	            END_IF;
	            IF NOT #iqUDT_WorkstationStatus."170".PEC_EoS.PEC THEN
	                IF #sa_TrackingArray_170[#iqUDT_Configuration."170".PEC_EoS.Distance / 10 - 2] > #iqUDT_Configuration.GlobalConfig.GINRangeStart
	                    AND #sa_TrackingArray_170[#iqUDT_Configuration."170".PEC_EoS.Distance / 10 - 2] < ((#iqUDT_Configuration.GlobalConfig.GINRangeStart + #iqUDT_Configuration.GlobalConfig.GINRangeEnd) / 2) THEN
	                    IF #si_EmptyBinRequiredCounter1X0 > 0 THEN
	                        #si_EmptyBinRequiredCounter1X0 -= 1;
	                    END_IF;
	                ELSE

	                    IF #si_PartialyBinRequiredCounter1X0 > 0 THEN
	                        #si_PartialyBinRequiredCounter1X0 -= 1;
	                    ELSE
	                        IF #si_EmptyBinRequiredCounter1X0 > 0 THEN
	                            #si_EmptyBinRequiredCounter1X0 -= 1;
	                        END_IF;


	                    END_IF;

	                END_IF;


	            END_IF; *)


	        END_REGION

	    END_REGION

	    REGION Barcode handling

	        REGION 050

	            IF #iqUDT_WorkstationCommonStatus."050".Dieback
	                AND NOT #iqUDT_WorkstationStatus."050".PEC_EoS.PEC
	                AND #sa_TrackingArray_050[(#iqUDT_Configuration."050".PEC_EoS.Distance / 10) - 1] > 0
	            THEN

	                IF #iqUDT_FirstWESInterface.Field[1].WES2PLC.SetContainerID THEN

	                    "DB_GIN".GIN[#sa_TrackingArray_050[(#iqUDT_Configuration."050".PEC_EoS.Distance / 10) - 1]].General.Identification.Barcode := #iqUDT_FirstWESInterface.Field[1].WES2PLC.ContainerID;
	                    #iqUDT_FirstWESInterface.Field[1].WES2PLC.SetContainerID := 0;

	                END_IF;

	                IF #iqUDT_FirstWESInterface.Field[1].PLC2WES.ContainerID <> "DB_GIN".GIN[#sa_TrackingArray_050[(#iqUDT_Configuration."050".PEC_EoS.Distance / 10) - 1]].General.Identification.Barcode
	                THEN

	                    #iqUDT_FirstWESInterface.Field[1].PLC2WES.ContainerID := "DB_GIN".GIN[#sa_TrackingArray_050[(#iqUDT_Configuration."050".PEC_EoS.Distance / 10) - 1]].General.Identification.Barcode;
	                    #iqUDT_FirstWESInterface.Field[1].PLC2WES.SetContainerID := TRUE;
	                END_IF;
	            ELSE
	                IF #iqUDT_FirstWESInterface.Field[1].PLC2WES.ContainerID <> #cs_MissingBarcodeCode
	                THEN
	                    #iqUDT_FirstWESInterface.Field[1].PLC2WES.ContainerID := #cs_MissingBarcodeCode;
	                    #iqUDT_FirstWESInterface.Field[1].PLC2WES.SetContainerID := TRUE;
	                END_IF;

	            END_IF;

	        END_REGION

	        REGION 060

	            IF #iqUDT_WorkstationCommonStatus."060".Dieback
	                AND NOT #iqUDT_WorkstationStatus."060".PEC_EoS.PEC
	                AND #sa_TrackingArray_060[(#iqUDT_Configuration."060".PEC_EoS.Distance / 10) - 1] > 0
	            THEN

	                IF #iqUDT_FirstWESInterface.Field[2].WES2PLC.SetContainerID THEN

	                    "DB_GIN".GIN[#sa_TrackingArray_060[(#iqUDT_Configuration."060".PEC_EoS.Distance / 10) - 1]].General.Identification.Barcode := #iqUDT_FirstWESInterface.Field[2].WES2PLC.ContainerID;
	                    #iqUDT_FirstWESInterface.Field[2].WES2PLC.SetContainerID := 0;

	                END_IF;

	                IF #iqUDT_FirstWESInterface.Field[2].PLC2WES.ContainerID <> "DB_GIN".GIN[#sa_TrackingArray_060[(#iqUDT_Configuration."060".PEC_EoS.Distance / 10) - 1]].General.Identification.Barcode
	                THEN

	                    #iqUDT_FirstWESInterface.Field[2].PLC2WES.ContainerID := "DB_GIN".GIN[#sa_TrackingArray_060[(#iqUDT_Configuration."060".PEC_EoS.Distance / 10) - 1]].General.Identification.Barcode;
	                    #iqUDT_FirstWESInterface.Field[2].PLC2WES.SetContainerID := TRUE;
	                END_IF;
	            ELSE
	                IF #iqUDT_FirstWESInterface.Field[2].PLC2WES.ContainerID <> #cs_MissingBarcodeCode
	                THEN
	                    #iqUDT_FirstWESInterface.Field[2].PLC2WES.ContainerID := #cs_MissingBarcodeCode;
	                    #iqUDT_FirstWESInterface.Field[2].PLC2WES.SetContainerID := TRUE;
	                END_IF;

	            END_IF;

	        END_REGION

	        REGION 070

	            IF #iqUDT_WorkstationCommonStatus."070".Dieback
	                AND NOT #iqUDT_WorkstationStatus."070".PEC_EoS.PEC
	                AND #sa_TrackingArray_070[(#iqUDT_Configuration."070".PEC_EoS.Distance / 10) - 1] > 0
	            THEN

	                IF #iqUDT_FirstWESInterface.Field[3].WES2PLC.SetContainerID THEN

	                    "DB_GIN".GIN[#sa_TrackingArray_070[(#iqUDT_Configuration."070".PEC_EoS.Distance / 10) - 1]].General.Identification.Barcode := #iqUDT_FirstWESInterface.Field[3].WES2PLC.ContainerID;
	                    #iqUDT_FirstWESInterface.Field[3].WES2PLC.SetContainerID := 0;

	                END_IF;

	                IF #iqUDT_FirstWESInterface.Field[3].PLC2WES.ContainerID <> "DB_GIN".GIN[#sa_TrackingArray_070[(#iqUDT_Configuration."070".PEC_EoS.Distance / 10) - 1]].General.Identification.Barcode
	                THEN

	                    #iqUDT_FirstWESInterface.Field[3].PLC2WES.ContainerID := "DB_GIN".GIN[#sa_TrackingArray_070[(#iqUDT_Configuration."070".PEC_EoS.Distance / 10) - 1]].General.Identification.Barcode;
	                    #iqUDT_FirstWESInterface.Field[3].PLC2WES.SetContainerID := TRUE;
	                END_IF;
	            ELSE
	                IF #iqUDT_FirstWESInterface.Field[3].PLC2WES.ContainerID <> #cs_MissingBarcodeCode
	                THEN
	                    #iqUDT_FirstWESInterface.Field[3].PLC2WES.ContainerID := #cs_MissingBarcodeCode;
	                    #iqUDT_FirstWESInterface.Field[3].PLC2WES.SetContainerID := TRUE;
	                END_IF;

	            END_IF;

	        END_REGION


	        REGION 150

	            IF #iqUDT_WorkstationCommonStatus."150".Dieback
	                AND NOT #iqUDT_WorkstationStatus."150".PEC_EoS.PEC
	                AND #sa_TrackingArray_150[(#iqUDT_Configuration."150".PEC_EoS.Distance / 10) - 1] > 0
	            THEN

	                IF #iqUDT_SecondWESInterface.Field[1].WES2PLC.SetContainerID THEN

	                    "DB_GIN".GIN[#sa_TrackingArray_150[(#iqUDT_Configuration."150".PEC_EoS.Distance / 10) - 1]].General.Identification.Barcode := #iqUDT_SecondWESInterface.Field[1].WES2PLC.ContainerID;
	                    #iqUDT_SecondWESInterface.Field[1].WES2PLC.SetContainerID := 0;

	                END_IF;

	                IF #iqUDT_SecondWESInterface.Field[1].PLC2WES.ContainerID <> "DB_GIN".GIN[#sa_TrackingArray_150[(#iqUDT_Configuration."150".PEC_EoS.Distance / 10) - 1]].General.Identification.Barcode
	                THEN

	                    #iqUDT_SecondWESInterface.Field[1].PLC2WES.ContainerID := "DB_GIN".GIN[#sa_TrackingArray_150[(#iqUDT_Configuration."150".PEC_EoS.Distance / 10) - 1]].General.Identification.Barcode;
	                    #iqUDT_SecondWESInterface.Field[1].PLC2WES.SetContainerID := TRUE;
	                END_IF;
	            ELSE
	                IF #iqUDT_SecondWESInterface.Field[1].PLC2WES.ContainerID <> #cs_MissingBarcodeCode
	                THEN
	                    #iqUDT_SecondWESInterface.Field[1].PLC2WES.ContainerID := #cs_MissingBarcodeCode;
	                    #iqUDT_SecondWESInterface.Field[1].PLC2WES.SetContainerID := TRUE;
	                END_IF;

	            END_IF;

	        END_REGION

	        REGION 160

	            IF #iqUDT_WorkstationCommonStatus."160".Dieback
	                AND NOT #iqUDT_WorkstationStatus."160".PEC_EoS.PEC
	                AND #sa_TrackingArray_160[(#iqUDT_Configuration."160".PEC_EoS.Distance / 10) - 1] > 0
	            THEN

	                IF #iqUDT_SecondWESInterface.Field[2].WES2PLC.SetContainerID THEN

	                    "DB_GIN".GIN[#sa_TrackingArray_160[(#iqUDT_Configuration."160".PEC_EoS.Distance / 10) - 1]].General.Identification.Barcode := #iqUDT_SecondWESInterface.Field[2].WES2PLC.ContainerID;
	                    #iqUDT_SecondWESInterface.Field[2].WES2PLC.SetContainerID := 0;

	                END_IF;

	                IF #iqUDT_SecondWESInterface.Field[2].PLC2WES.ContainerID <> "DB_GIN".GIN[#sa_TrackingArray_160[(#iqUDT_Configuration."160".PEC_EoS.Distance / 10) - 1]].General.Identification.Barcode
	                THEN

	                    #iqUDT_SecondWESInterface.Field[2].PLC2WES.ContainerID := "DB_GIN".GIN[#sa_TrackingArray_160[(#iqUDT_Configuration."160".PEC_EoS.Distance / 10) - 1]].General.Identification.Barcode;
	                    #iqUDT_SecondWESInterface.Field[2].PLC2WES.SetContainerID := TRUE;
	                END_IF;
	            ELSE
	                IF #iqUDT_SecondWESInterface.Field[2].PLC2WES.ContainerID <> #cs_MissingBarcodeCode
	                THEN
	                    #iqUDT_SecondWESInterface.Field[2].PLC2WES.ContainerID := #cs_MissingBarcodeCode;
	                    #iqUDT_SecondWESInterface.Field[2].PLC2WES.SetContainerID := TRUE;
	                END_IF;

	            END_IF;

	        END_REGION

	        REGION 170

	            IF #iqUDT_WorkstationCommonStatus."170".Dieback
	                AND NOT #iqUDT_WorkstationStatus."170".PEC_EoS.PEC
	                AND #sa_TrackingArray_170[(#iqUDT_Configuration."170".PEC_EoS.Distance / 10) - 1] > 0
	            THEN

	                IF #iqUDT_SecondWESInterface.Field[3].WES2PLC.SetContainerID THEN

	                    "DB_GIN".GIN[#sa_TrackingArray_170[(#iqUDT_Configuration."170".PEC_EoS.Distance / 10) - 1]].General.Identification.Barcode := #iqUDT_SecondWESInterface.Field[3].WES2PLC.ContainerID;
	                    #iqUDT_SecondWESInterface.Field[3].WES2PLC.SetContainerID := 0;

	                END_IF;

	                IF #iqUDT_SecondWESInterface.Field[3].PLC2WES.ContainerID <> "DB_GIN".GIN[#sa_TrackingArray_170[(#iqUDT_Configuration."170".PEC_EoS.Distance / 10) - 1]].General.Identification.Barcode
	                THEN

	                    #iqUDT_SecondWESInterface.Field[3].PLC2WES.ContainerID := "DB_GIN".GIN[#sa_TrackingArray_170[(#iqUDT_Configuration."170".PEC_EoS.Distance / 10) - 1]].General.Identification.Barcode;
	                    #iqUDT_SecondWESInterface.Field[3].PLC2WES.SetContainerID := TRUE;
	                END_IF;
	            ELSE
	                IF #iqUDT_SecondWESInterface.Field[3].PLC2WES.ContainerID <> #cs_MissingBarcodeCode
	                THEN
	                    #iqUDT_SecondWESInterface.Field[3].PLC2WES.ContainerID := #cs_MissingBarcodeCode;
	                    #iqUDT_SecondWESInterface.Field[3].PLC2WES.SetContainerID := TRUE;
	                END_IF;

	            END_IF;

	        END_REGION


	    END_REGION

	    REGION Clearing tracking

	        IF (#sx_Hold050
	            AND #sa_TrackingArray_050[(#iqUDT_Configuration."050".PEC_EoS.Distance - 10) / 10] <> 0
	            AND #iqUDT_WorkstationStatus."050".PEC_EoS.PEC)

	        THEN

	            #tx_ArraySize := "FC_GetNrOfArrayEl"(#sa_TrackingArray_050);

	            FILL_BLK(IN    := 0,
	                     COUNT := INT_TO_ULINT(#tx_ArraySize),
	                     OUT   => #sa_TrackingArray_050[0]);

	        END_IF;

	        IF (#sx_Hold060
	            AND #sa_TrackingArray_060[(#iqUDT_Configuration."060".PEC_EoS.Distance - 10) / 10] <> 0
	            AND #iqUDT_WorkstationStatus."060".PEC_EoS.PEC)

	        THEN

	            #tx_ArraySize := "FC_GetNrOfArrayEl"(#sa_TrackingArray_060);

	            FILL_BLK(IN    := 0,
	                     COUNT := INT_TO_ULINT(#tx_ArraySize),
	                     OUT   => #sa_TrackingArray_060[0]);

	        END_IF;

	        IF (#sx_Hold070
	            AND #sa_TrackingArray_070[(#iqUDT_Configuration."070".PEC_EoS.Distance - 10) / 10] <> 0
	            AND #iqUDT_WorkstationStatus."070".PEC_EoS.PEC)

	        THEN

	            #tx_ArraySize := "FC_GetNrOfArrayEl"(#sa_TrackingArray_070);

	            FILL_BLK(IN    := 0,
	                     COUNT := INT_TO_ULINT(#tx_ArraySize),
	                     OUT   => #sa_TrackingArray_070[0]);

	        END_IF;


	        IF (#sx_Hold150
	            AND #sa_TrackingArray_150[(#iqUDT_Configuration."150".PEC_EoS.Distance - 10) / 10] <> 0
	            AND #iqUDT_WorkstationStatus."150".PEC_EoS.PEC)

	        THEN

	            #tx_ArraySize := "FC_GetNrOfArrayEl"(#sa_TrackingArray_150);

	            FILL_BLK(IN    := 0,
	                     COUNT := INT_TO_ULINT(#tx_ArraySize),
	                     OUT   => #sa_TrackingArray_150[0]);

	        END_IF;

	        IF (#sx_Hold160
	            AND #sa_TrackingArray_160[(#iqUDT_Configuration."160".PEC_EoS.Distance - 10) / 10] <> 0
	            AND #iqUDT_WorkstationStatus."160".PEC_EoS.PEC)

	        THEN

	            #tx_ArraySize := "FC_GetNrOfArrayEl"(#sa_TrackingArray_160);

	            FILL_BLK(IN    := 0,
	                     COUNT := INT_TO_ULINT(#tx_ArraySize),
	                     OUT   => #sa_TrackingArray_060[0]);

	        END_IF;

	        IF (#sx_Hold170
	            AND #sa_TrackingArray_170[(#iqUDT_Configuration."170".PEC_EoS.Distance - 10) / 10] <> 0
	            AND #iqUDT_WorkstationStatus."170".PEC_EoS.PEC)

	        THEN

	            #tx_ArraySize := "FC_GetNrOfArrayEl"(#sa_TrackingArray_170);

	            FILL_BLK(IN    := 0,
	                     COUNT := INT_TO_ULINT(#tx_ArraySize),
	                     OUT   => #sa_TrackingArray_170[0]);

	        END_IF;

	    END_REGION


	    REGION Buffer state

	        #sFB_Pulse_UpdateBufferState(iudi_PulseTime := #cudi_UpdateBufferState);

	        IF #sFB_Pulse_UpdateBufferState.qx_Pulse THEN

	            #sFB_CountActiveInputs(ix_Input1            := NOT #iqUDT_WorkstationStatus."010".PEC_EoS.PEC,
	                                   ix_Input2            := NOT #iqUDT_WorkstationStatus."020".PEC_EoS.PEC,
	                                   ix_Input3            := NOT #iqUDT_WorkstationStatus."030".PEC_EoS.PEC,
	                                   ix_Input4            := FALSE,
	                                   ix_Input5            := FALSE,
	                                   ix_Input6            := FALSE,
	                                   ix_Input7            := FALSE,
	                                   ix_Input8            := FALSE,
	                                   ix_Input9            := FALSE,
	                                   ix_Input10           := FALSE,
	                                   ix_Input11           := FALSE,
	                                   ix_Input12           := FALSE,
	                                   ix_Input13           := FALSE,
	                                   ix_Input14           := FALSE,
	                                   ix_Input15           := FALSE,
	                                   ix_Input16           := FALSE,
	                                   qi_ActiveInputsCount => #qi_FirstBufferState);


	            #sFB_CountActiveInputs(ix_Input1            := NOT #iqUDT_WorkstationStatus."110".PEC_EoS.PEC,
	                                   ix_Input2            := NOT #iqUDT_WorkstationStatus."120".PEC_EoS.PEC,
	                                   ix_Input3            := NOT #iqUDT_WorkstationStatus."130".PEC_EoS.PEC,
	                                   ix_Input4            := FALSE,
	                                   ix_Input5            := FALSE,
	                                   ix_Input6            := FALSE,
	                                   ix_Input7            := FALSE,
	                                   ix_Input8            := FALSE,
	                                   ix_Input9            := FALSE,
	                                   ix_Input10           := FALSE,
	                                   ix_Input11           := FALSE,
	                                   ix_Input12           := FALSE,
	                                   ix_Input13           := FALSE,
	                                   ix_Input14           := FALSE,
	                                   ix_Input15           := FALSE,
	                                   ix_Input16           := FALSE,
	                                   qi_ActiveInputsCount => #qi_SecondBufferState);

	        END_IF;



	    END_REGION


	    REGION Finish operation

	        #sF_TRIG_ParcelArrived0X0(CLK := #iqUDT_WorkstationStatus."050".PEC_EoS.PEC);
	        #sF_TRIG_ParcelArrived1X0(CLK := #iqUDT_WorkstationStatus."150".PEC_EoS.PEC);
	        #sF_TRIG_ParcelArrived2X0(CLK := #iqUDT_WorkstationStatus."250".PEC_EoS.PEC);

	        // Check if operation if finished. If yes then set operation in progress bit
	        IF #si_SendTo0X0 AND (#sF_TRIG_ParcelArrived0X0.Q OR #sFB_TimerOnOffDelay_OperationTimeout.qx_DelayedSignal) THEN

	            #si_SendTo0X0 := FALSE;

	        END_IF;


	        IF #si_SendTo1X0 AND (#sF_TRIG_ParcelArrived1X0.Q OR #sFB_TimerOnOffDelay_OperationTimeout.qx_DelayedSignal) THEN

	            #si_SendTo1X0 := FALSE;

	        END_IF;

	        IF #si_SendTo2X0 AND (#sF_TRIG_ParcelArrived2X0.Q OR #sFB_TimerOnOffDelay_OperationTimeout.qx_DelayedSignal) THEN

	            #si_SendTo2X0 := FALSE;

	        END_IF;


	        IF NOT #si_SendTo0X0 AND NOT #si_SendTo1X0 AND NOT #si_SendTo2X0
	            AND #sUDT_Interface_040.ActualSpeed = 0
	            AND #sUDT_Interface_041.ActualSpeed = 0
	            AND #sUDT_Interface_140.ActualSpeed = 0
	            AND #sUDT_Interface_141.ActualSpeed = 0
	            AND #sUDT_Interface_240.ActualSpeed = 0
	            AND #sUDT_Interface_241.ActualSpeed = 0
	        THEN

	            #sx_NoOperationInProgress := TRUE;
	            #si_040DestinationA := 0;
	            #si_040DestinationB := 0;
	            #si_040DestinationC := 0;
	            #si_040DestinationD := 0;

	            #si_140DestinationA := 0;
	            #si_140DestinationB := 0;
	            #si_140DestinationC := 0;
	            #si_140DestinationD := 0;

	            #si_240DestinationA := 0;
	            #si_240DestinationB := 0;
	            #si_240DestinationC := 0;
	            #si_240DestinationD := 0;

	            #sx_Hold030 := FALSE;
	            #sx_Hold130 := FALSE;
	            #sx_Hold020 := FALSE;
	            #sx_Hold120 := FALSE;
	            #sx_Hold230 := FALSE;
	            #sx_Hold220 := FALSE;

	            #sx_Hold050 := TRUE;
	            #sx_Hold060 := TRUE;
	            #sx_Hold070 := TRUE;

	            #sx_Hold150 := TRUE;
	            #sx_Hold160 := TRUE;
	            #sx_Hold170 := TRUE;

	            #sx_Enable0X0In := FALSE;
	            #sx_Enable1X0In := FALSE;
	            #sx_Enable2X0In := FALSE;

	        END_IF;


	    END_REGION

	    (*
	    REGION Workstation initialization

	        #sR_TRIG_InitializeFirstWS(CLK := #sx_FirstStationActive);

	        IF #sR_TRIG_InitializeFirstWS.Q THEN

	            #sx_StartClearing := FALSE;
	            IF #iqUDT_WorkstationStatus."010".PEC_EoS.PEC THEN

	                #si_ReqestNewEmptyBin += 1;

	            END_IF;

	            IF #iqUDT_WorkstationStatus."020".PEC_EoS.PEC THEN

	                #si_ReqestNewEmptyBin += 1;

	            END_IF;

	            IF #iqUDT_WorkstationStatus."030".PEC_EoS.PEC THEN

	                #si_ReqestNewEmptyBin += 1;

	            END_IF;


	            (*
	            #si_EmptyBinRequiredCounter0X0 := 2;
	            #si_PartialyBinRequiredCounter0X0 := 1;


	            REGION 050 Workposition initialization
	                IF NOT #iqUDT_WorkstationStatus."050".PEC_EoS.PEC THEN
	                    IF #sa_TrackingArray_050[#iqUDT_Configuration."050".PEC_EoS.Distance / 10 - 2] > #iqUDT_Configuration.GlobalConfig.GINRangeStart
	                        AND #sa_TrackingArray_050[#iqUDT_Configuration."050".PEC_EoS.Distance / 10 - 2] < ((#iqUDT_Configuration.GlobalConfig.GINRangeStart + #iqUDT_Configuration.GlobalConfig.GINRangeEnd) / 2) THEN
	                        IF #si_EmptyBinRequiredCounter0X0 > 0 THEN
	                            #si_EmptyBinRequiredCounter0X0 -= 1;
	                        END_IF;
	                    ELSE

	                        IF #si_PartialyBinRequiredCounter0X0 > 0 THEN
	                            #si_PartialyBinRequiredCounter0X0 -= 1;
	                        ELSE
	                            IF #si_EmptyBinRequiredCounter0X0 > 0 THEN
	                                #si_EmptyBinRequiredCounter0X0 -= 1;
	                            END_IF;


	                        END_IF;

	                    END_IF;


	                END_IF;
	            END_REGION

	            REGION 060 Workposition initialization
	                IF NOT #iqUDT_WorkstationStatus."060".PEC_EoS.PEC THEN
	                    IF #sa_TrackingArray_060[#iqUDT_Configuration."060".PEC_EoS.Distance / 10 - 2] > #iqUDT_Configuration.GlobalConfig.GINRangeStart
	                        AND #sa_TrackingArray_060[#iqUDT_Configuration."060".PEC_EoS.Distance / 10 - 2] < ((#iqUDT_Configuration.GlobalConfig.GINRangeStart + #iqUDT_Configuration.GlobalConfig.GINRangeEnd) / 2) THEN
	                        IF #si_EmptyBinRequiredCounter0X0 > 0 THEN
	                            #si_EmptyBinRequiredCounter0X0 -= 1;
	                        END_IF;
	                    ELSE

	                        IF #si_PartialyBinRequiredCounter0X0 > 0 THEN
	                            #si_PartialyBinRequiredCounter0X0 -= 1;
	                        ELSE
	                            IF #si_EmptyBinRequiredCounter0X0 > 0 THEN
	                                #si_EmptyBinRequiredCounter0X0 -= 1;
	                            END_IF;


	                        END_IF;

	                    END_IF;


	                END_IF;
	            END_REGION

	            REGION 070 Workposition initialization
	                IF NOT #iqUDT_WorkstationStatus."070".PEC_EoS.PEC THEN
	                    IF #sa_TrackingArray_070[#iqUDT_Configuration."070".PEC_EoS.Distance / 10 - 2] > #iqUDT_Configuration.GlobalConfig.GINRangeStart
	                        AND #sa_TrackingArray_070[#iqUDT_Configuration."070".PEC_EoS.Distance / 10 - 2] < ((#iqUDT_Configuration.GlobalConfig.GINRangeStart + #iqUDT_Configuration.GlobalConfig.GINRangeEnd) / 2) THEN
	                        IF #si_EmptyBinRequiredCounter0X0 > 0 THEN
	                            #si_EmptyBinRequiredCounter0X0 -= 1;
	                        END_IF;
	                    ELSE

	                        IF #si_PartialyBinRequiredCounter0X0 > 0 THEN
	                            #si_PartialyBinRequiredCounter0X0 -= 1;
	                        ELSE
	                            IF #si_EmptyBinRequiredCounter0X0 > 0 THEN
	                                #si_EmptyBinRequiredCounter0X0 -= 1;
	                            END_IF;


	                        END_IF;

	                    END_IF;


	                END_IF;
	            END_REGION
	            *)

	        END_IF;

	        #sR_TRIG_InitializeSecondWS(CLK := #sx_SecondStationActive);

	        IF #sR_TRIG_InitializeSecondWS.Q THEN

	            IF #iqUDT_WorkstationStatus."110".PEC_EoS.PEC THEN

	                #si_ReqestNewPartialBin += 1;

	            END_IF;

	            IF #iqUDT_WorkstationStatus."120".PEC_EoS.PEC THEN

	                #si_ReqestNewPartialBin += 1;

	            END_IF;

	            IF #iqUDT_WorkstationStatus."130".PEC_EoS.PEC THEN

	                #si_ReqestNewPartialBin += 1;

	            END_IF;
	            (*
	            #si_EmptyBinRequiredCounter1X0 := 2;
	            #si_PartialyBinRequiredCounter1X0 := 1;

	             REGION 150 Workposition initialization
	                IF NOT #iqUDT_WorkstationStatus."150".PEC_EoS.PEC
	                THEN
	                    IF (#sa_TrackingArray_150[#iqUDT_Configuration."150".PEC_EoS.Distance / 10 / 10 - 2] > #iqUDT_Configuration.GlobalConfig.GINRangeStart
	                        AND #sa_TrackingArray_150[#iqUDT_Configuration."150".PEC_EoS.Distance / 10 - 2] < ((#iqUDT_Configuration.GlobalConfig.GINRangeStart + #iqUDT_Configuration.GlobalConfig.GINRangeEnd) / 2))
	                    THEN
	                        IF #si_EmptyBinRequiredCounter1X0 > 0 THEN
	                            #si_EmptyBinRequiredCounter1X0 -= 1;
	                        END_IF;
	                    ELSE

	                        IF #si_PartialyBinRequiredCounter1X0 > 0 THEN
	                            #si_PartialyBinRequiredCounter1X0 -= 1;
	                        ELSE
	                            IF #si_EmptyBinRequiredCounter1X0 > 0 THEN
	                                #si_EmptyBinRequiredCounter1X0 -= 1;
	                            END_IF;


	                        END_IF;

	                    END_IF;


	                END_IF;
	            END_REGION

	            REGION 160 Workposition initialization
	                IF NOT #iqUDT_WorkstationStatus."160".PEC_EoS.PEC THEN
	                    IF #sa_TrackingArray_160[#iqUDT_Configuration."160".PEC_EoS.Distance / 10 - 2] > #iqUDT_Configuration.GlobalConfig.GINRangeStart
	                        AND #sa_TrackingArray_160[#iqUDT_Configuration."160".PEC_EoS.Distance / 10 - 2] < ((#iqUDT_Configuration.GlobalConfig.GINRangeStart + #iqUDT_Configuration.GlobalConfig.GINRangeEnd) / 2) THEN
	                        IF #si_EmptyBinRequiredCounter1X0 > 0 THEN
	                            #si_EmptyBinRequiredCounter1X0 -= 1;
	                        END_IF;
	                    ELSE

	                        IF #si_PartialyBinRequiredCounter1X0 > 0 THEN
	                            #si_PartialyBinRequiredCounter1X0 -= 1;
	                        ELSE
	                            IF #si_EmptyBinRequiredCounter1X0 > 0 THEN
	                                #si_EmptyBinRequiredCounter1X0 -= 1;
	                            END_IF;


	                        END_IF;

	                    END_IF;


	                END_IF;
	            END_REGION

	            REGION 170 Workposition initialization
	                IF NOT #iqUDT_WorkstationStatus."170".PEC_EoS.PEC THEN
	                    IF #sa_TrackingArray_170[#iqUDT_Configuration."170".PEC_EoS.Distance / 10 - 2] > #iqUDT_Configuration.GlobalConfig.GINRangeStart
	                        AND #sa_TrackingArray_170[#iqUDT_Configuration."170".PEC_EoS.Distance / 10 - 2] < ((#iqUDT_Configuration.GlobalConfig.GINRangeStart + #iqUDT_Configuration.GlobalConfig.GINRangeEnd) / 2) THEN
	                        IF #si_EmptyBinRequiredCounter1X0 > 0 THEN
	                            #si_EmptyBinRequiredCounter1X0 -= 1;
	                        END_IF;
	                    ELSE

	                        IF #si_PartialyBinRequiredCounter1X0 > 0 THEN
	                            #si_PartialyBinRequiredCounter1X0 -= 1;
	                        ELSE
	                            IF #si_EmptyBinRequiredCounter1X0 > 0 THEN
	                                #si_EmptyBinRequiredCounter1X0 -= 1;
	                            END_IF;


	                        END_IF;

	                    END_IF;


	                END_IF;

	            END_REGION *)

	        END_IF;

	    END_REGION
	    *)
	    (*
	    REGION Request empty bin to buffer

	        IF #si_ReqestNewEmptyBin > 0 THEN

	            #ti_NumberOfBinInQueue := 0;
	            IF #iqUDT_EmptyBuffer.BufferState1.BinRequest THEN
	                #ti_NumberOfBinInQueue += 1;
	            END_IF;
	            IF #iqUDT_EmptyBuffer.BufferState2.BinRequest THEN
	                #ti_NumberOfBinInQueue += 1;
	            END_IF;
	            IF #iqUDT_EmptyBuffer.BufferState3.BinRequest THEN
	                #ti_NumberOfBinInQueue += 1;
	            END_IF;
	            IF NOT #iqUDT_WorkstationStatus."010".PEC_EoS.PEC THEN
	                #ti_NumberOfBinInQueue += 1;
	            END_IF;
	            IF NOT #iqUDT_WorkstationStatus."020".PEC_EoS.PEC THEN
	                #ti_NumberOfBinInQueue += 1;
	            END_IF;
	            IF NOT #iqUDT_WorkstationStatus."030".PEC_EoS.PEC THEN
	                #ti_NumberOfBinInQueue += 1;
	            END_IF;

	            IF #ti_NumberOfBinInQueue < 3 THEN

	                "FC_Fifo"(ic_Mode          := 'S',
	                          qUDT_Status      => #tUDT_FifoStatusEmpty,
	                          qx_Error         => #tx_Error,
	                          qx_Warning       => #tx_Warning,
	                          iqv_Data         := #iqUDT_Configuration.GlobalConfig.DestinationEmpty,
	                          iqUDT_FifoHeader := #iqa_EmptyFifoHeader,
	                          iqv_DataBuffer   := #iqa_EmptyFifoData);

	                IF NOT #tUDT_FifoStatusEmpty.FifoFull THEN

	                    "FC_Fifo"(ic_Mode          := 'W',
	                              qUDT_Status      => #tUDT_FifoStatusEmpty,
	                              qx_Error         => #tx_Error,
	                              qx_Warning       => #tx_Warning,
	                              iqv_Data         := #iqUDT_Configuration.GlobalConfig.DestinationEmpty,
	                              iqUDT_FifoHeader := #iqa_EmptyFifoHeader,
	                              iqv_DataBuffer   := #iqa_EmptyFifoData);

	                    IF NOT #iqUDT_EmptyBuffer.BufferState1.BinRequest THEN
	                        #iqUDT_EmptyBuffer.BufferState1.BinRequest := TRUE;
	                    ELSIF NOT #iqUDT_EmptyBuffer.BufferState2.BinRequest THEN
	                        #iqUDT_EmptyBuffer.BufferState2.BinRequest := TRUE;
	                    ELSE
	                        #iqUDT_EmptyBuffer.BufferState3.BinRequest := TRUE;
	                    END_IF;

	                    #si_ReqestNewEmptyBin -= 1;
	                    #iqUDT_EmptyBuffer.Destination := #iqUDT_Configuration.GlobalConfig.DestinationEmpty;
	                END_IF;



	            END_IF;

	        END_IF;


	    END_REGION
	    *)
	    (*
	    REGION Request partial bin to buffer

	        IF #si_ReqestNewPartialBin > 0 THEN

	            #ti_NumberOfBinInQueue := 0;
	            IF #iqUDT_PartialBuffer.BufferState1.BinRequest THEN
	                #ti_NumberOfBinInQueue += 1;
	            END_IF;
	            IF #iqUDT_PartialBuffer.BufferState2.BinRequest THEN
	                #ti_NumberOfBinInQueue += 1;
	            END_IF;
	            IF #iqUDT_PartialBuffer.BufferState3.BinRequest THEN
	                #ti_NumberOfBinInQueue += 1;
	            END_IF;
	            IF NOT #iqUDT_WorkstationStatus."110".PEC_EoS.PEC THEN
	                #ti_NumberOfBinInQueue += 1;
	            END_IF;
	            IF NOT #iqUDT_WorkstationStatus."120".PEC_EoS.PEC THEN
	                #ti_NumberOfBinInQueue += 1;
	            END_IF;
	            IF NOT #iqUDT_WorkstationStatus."130".PEC_EoS.PEC THEN
	                #ti_NumberOfBinInQueue += 1;
	            END_IF;

	            IF #ti_NumberOfBinInQueue < 3 THEN



	                "FC_Fifo"(ic_Mode          := 'S',
	                          qUDT_Status      => #tUDT_FifoStatusPartial,
	                          qx_Error         => #tx_Error,
	                          qx_Warning       => #tx_Warning,
	                          iqv_Data         := #iqUDT_Configuration.GlobalConfig.DestinationPartialy,
	                          iqUDT_FifoHeader := #iqa_PartialFifoHeader,
	                          iqv_DataBuffer   := #iqa_PartialFifoData);

	                IF NOT #tUDT_FifoStatusPartial.FifoFull THEN

	                    "FC_Fifo"(ic_Mode          := 'W',
	                              qUDT_Status      => #tUDT_FifoStatusPartial,
	                              qx_Error         => #tx_Error,
	                              qx_Warning       => #tx_Warning,
	                              iqv_Data         := #iqUDT_Configuration.GlobalConfig.DestinationPartialy,
	                              iqUDT_FifoHeader := #iqa_PartialFifoHeader,
	                              iqv_DataBuffer   := #iqa_PartialFifoData);

	                    IF NOT #iqUDT_PartialBuffer.BufferState1.BinRequest THEN
	                        #iqUDT_PartialBuffer.BufferState1.BinRequest := TRUE;
	                    ELSIF NOT #iqUDT_PartialBuffer.BufferState2.BinRequest THEN
	                        #iqUDT_PartialBuffer.BufferState2.BinRequest := TRUE;
	                    ELSE
	                        #iqUDT_PartialBuffer.BufferState3.BinRequest := TRUE;
	                    END_IF;

	                    #si_ReqestNewPartialBin -= 1;
	                    #iqUDT_PartialBuffer.Destination := #iqUDT_Configuration.GlobalConfig.DestinationPartialy;

	                END_IF;

	            END_IF;

	        END_IF;

	    END_REGION
	    *)
	    (*
	    REGION Ordered bin monitoring

	        IF "DB_Memory".OS_2sec THEN

	            IF #iqUDT_EmptyBuffer.BufferState1.BinSend THEN
	                #iqUDT_EmptyBuffer.BufferState1.WaintingTime += 2;

	                IF #iqUDT_EmptyBuffer.BufferState1.WaintingTime > #iqUDT_Configuration.GlobalConfig.BinOrderTimeout THEN

	                    #iqUDT_EmptyBuffer.BufferState1 := #iqUDT_EmptyBuffer.BufferState2;
	                    #iqUDT_EmptyBuffer.BufferState2 := #iqUDT_EmptyBuffer.BufferState3;

	                    #iqUDT_EmptyBuffer.BufferState3.BinSend := FALSE;
	                    #iqUDT_EmptyBuffer.BufferState3.BinRequest := FALSE;
	                    #iqUDT_EmptyBuffer.BufferState3.UpcomingBarcode := '';
	                    #iqUDT_EmptyBuffer.BufferState3.WaintingTime := 0;


	                    #ti_NumberOfBinInQueue := 0;
	                    IF #iqUDT_EmptyBuffer.BufferState1.BinRequest THEN
	                        #ti_NumberOfBinInQueue += 1;
	                    END_IF;
	                    IF #iqUDT_EmptyBuffer.BufferState2.BinRequest THEN
	                        #ti_NumberOfBinInQueue += 1;
	                    END_IF;
	                    IF NOT #iqUDT_WorkstationStatus."010".PEC_EoS.PEC THEN
	                        #ti_NumberOfBinInQueue += 1;
	                    END_IF;
	                    IF NOT #iqUDT_WorkstationStatus."020".PEC_EoS.PEC THEN
	                        #ti_NumberOfBinInQueue += 1;
	                    END_IF;
	                    IF NOT #iqUDT_WorkstationStatus."030".PEC_EoS.PEC THEN
	                        #ti_NumberOfBinInQueue += 1;
	                    END_IF;

	                    IF #ti_NumberOfBinInQueue < 3 THEN
	                        #si_ReqestNewEmptyBin += 1;
	                    END_IF;


	                END_IF;

	            END_IF;

	            IF #iqUDT_EmptyBuffer.BufferState2.BinSend THEN
	                #iqUDT_EmptyBuffer.BufferState2.WaintingTime += 2;

	                IF #iqUDT_EmptyBuffer.BufferState2.WaintingTime > #iqUDT_Configuration.GlobalConfig.BinOrderTimeout THEN

	                    #iqUDT_EmptyBuffer.BufferState2 := #iqUDT_EmptyBuffer.BufferState3;

	                    #iqUDT_EmptyBuffer.BufferState3.BinSend := FALSE;
	                    #iqUDT_EmptyBuffer.BufferState3.BinRequest := FALSE;
	                    #iqUDT_EmptyBuffer.BufferState3.UpcomingBarcode := '';
	                    #iqUDT_EmptyBuffer.BufferState3.WaintingTime := 0;

	                    #si_ReqestNewEmptyBin += 1;

	                END_IF;

	            END_IF;

	            IF #iqUDT_EmptyBuffer.BufferState3.BinSend THEN
	                #iqUDT_EmptyBuffer.BufferState3.WaintingTime += 2;

	                IF #iqUDT_EmptyBuffer.BufferState3.WaintingTime > #iqUDT_Configuration.GlobalConfig.BinOrderTimeout THEN

	                    #iqUDT_EmptyBuffer.BufferState3.BinSend := FALSE;
	                    #iqUDT_EmptyBuffer.BufferState3.BinRequest := FALSE;
	                    #iqUDT_EmptyBuffer.BufferState3.UpcomingBarcode := '';
	                    #iqUDT_EmptyBuffer.BufferState3.WaintingTime := 0;
	                    #si_ReqestNewEmptyBin += 1;

	                END_IF;

	            END_IF;

	            IF #iqUDT_PartialBuffer.BufferState1.BinSend THEN
	                #iqUDT_PartialBuffer.BufferState1.WaintingTime += 2;

	                IF #iqUDT_PartialBuffer.BufferState1.WaintingTime > #iqUDT_Configuration.GlobalConfig.BinOrderTimeout THEN

	                    #iqUDT_PartialBuffer.BufferState1 := #iqUDT_PartialBuffer.BufferState2;
	                    #iqUDT_PartialBuffer.BufferState2 := #iqUDT_PartialBuffer.BufferState3;
	                    #iqUDT_PartialBuffer.BufferState3.BinSend := FALSE;
	                    #iqUDT_PartialBuffer.BufferState3.BinRequest := FALSE;
	                    #iqUDT_PartialBuffer.BufferState3.UpcomingBarcode := '';
	                    #iqUDT_PartialBuffer.BufferState3.WaintingTime := 0;


	                    #ti_NumberOfBinInQueue := 0;
	                    IF #iqUDT_PartialBuffer.BufferState1.BinRequest THEN
	                        #ti_NumberOfBinInQueue += 1;
	                    END_IF;
	                    IF #iqUDT_PartialBuffer.BufferState2.BinRequest THEN
	                        #ti_NumberOfBinInQueue += 1;
	                    END_IF;
	                    IF NOT #iqUDT_WorkstationStatus."110".PEC_EoS.PEC THEN
	                        #ti_NumberOfBinInQueue += 1;
	                    END_IF;
	                    IF NOT #iqUDT_WorkstationStatus."120".PEC_EoS.PEC THEN
	                        #ti_NumberOfBinInQueue += 1;
	                    END_IF;
	                    IF NOT #iqUDT_WorkstationStatus."130".PEC_EoS.PEC THEN
	                        #ti_NumberOfBinInQueue += 1;
	                    END_IF;

	                    IF #ti_NumberOfBinInQueue < 3 THEN
	                        #si_ReqestNewPartialBin += 1;
	                    END_IF;

	                END_IF;

	            END_IF;


	            IF #iqUDT_PartialBuffer.BufferState2.BinSend THEN
	                #iqUDT_PartialBuffer.BufferState2.WaintingTime += 2;
	                IF #iqUDT_PartialBuffer.BufferState2.WaintingTime > #iqUDT_Configuration.GlobalConfig.BinOrderTimeout THEN

	                    #iqUDT_PartialBuffer.BufferState2 := #iqUDT_PartialBuffer.BufferState3;

	                    #iqUDT_PartialBuffer.BufferState3.BinSend := FALSE;
	                    #iqUDT_PartialBuffer.BufferState3.BinRequest := FALSE;
	                    #iqUDT_PartialBuffer.BufferState3.UpcomingBarcode := '';
	                    #iqUDT_PartialBuffer.BufferState3.WaintingTime := 0;

	                    #si_ReqestNewPartialBin += 1;

	                END_IF;

	            END_IF;

	            IF #iqUDT_PartialBuffer.BufferState3.BinSend THEN
	                #iqUDT_PartialBuffer.BufferState3.WaintingTime += 2;

	                IF #iqUDT_PartialBuffer.BufferState3.WaintingTime > #iqUDT_Configuration.GlobalConfig.BinOrderTimeout THEN

	                    #iqUDT_PartialBuffer.BufferState3.BinSend := FALSE;
	                    #iqUDT_PartialBuffer.BufferState3.BinRequest := FALSE;
	                    #iqUDT_PartialBuffer.BufferState3.UpcomingBarcode := '';
	                    #iqUDT_PartialBuffer.BufferState3.WaintingTime := 0;
	                    #si_ReqestNewPartialBin += 1;

	                END_IF;
	            END_IF;

	        END_IF;

	    END_REGION
	    *)
	    (*
	    REGION Ordered product confirmation

	        REGION Empty

	            #sR_TRIG_EmptyBinReceived(CLK := #sa_TrackingArray_010[#iqUDT_Configuration."010".PEC_EoS.Distance / 10 - 1] <> 0);

	            IF #sR_TRIG_EmptyBinReceived.Q THEN

	                IF #iqUDT_EmptyBuffer.BufferState1.BinSend AND "DB_GIN".GIN[#sa_TrackingArray_010[#iqUDT_Configuration."010".PEC_EoS.Distance / 10 - 1]].General.Identification.Barcode = #iqUDT_EmptyBuffer.BufferState1.UpcomingBarcode THEN

	                    #iqUDT_EmptyBuffer.BufferState1 := #iqUDT_EmptyBuffer.BufferState2;
	                    #iqUDT_EmptyBuffer.BufferState2 := #iqUDT_EmptyBuffer.BufferState3;

	                    #iqUDT_EmptyBuffer.BufferState3.BinSend := FALSE;
	                    #iqUDT_EmptyBuffer.BufferState3.BinRequest := FALSE;
	                    #iqUDT_EmptyBuffer.BufferState3.UpcomingBarcode := '';
	                    #iqUDT_EmptyBuffer.BufferState3.WaintingTime := 0;
	                END_IF;


	                IF #iqUDT_EmptyBuffer.BufferState2.BinSend AND "DB_GIN".GIN[#sa_TrackingArray_010[#iqUDT_Configuration."010".PEC_EoS.Distance / 10 - 1]].General.Identification.Barcode = #iqUDT_EmptyBuffer.BufferState2.UpcomingBarcode THEN

	                    #iqUDT_EmptyBuffer.BufferState2 := #iqUDT_EmptyBuffer.BufferState3;

	                    #iqUDT_EmptyBuffer.BufferState3.BinSend := FALSE;
	                    #iqUDT_EmptyBuffer.BufferState3.BinRequest := FALSE;
	                    #iqUDT_EmptyBuffer.BufferState3.UpcomingBarcode := '';
	                    #iqUDT_EmptyBuffer.BufferState3.WaintingTime := 0;
	                END_IF;


	                IF #iqUDT_EmptyBuffer.BufferState3.BinSend AND "DB_GIN".GIN[#sa_TrackingArray_010[#iqUDT_Configuration."010".PEC_EoS.Distance / 10 - 1]].General.Identification.Barcode = #iqUDT_EmptyBuffer.BufferState3.UpcomingBarcode THEN

	                    #iqUDT_EmptyBuffer.BufferState3.BinSend := FALSE;
	                    #iqUDT_EmptyBuffer.BufferState3.BinRequest := FALSE;
	                    #iqUDT_EmptyBuffer.BufferState3.UpcomingBarcode := '';
	                    #iqUDT_EmptyBuffer.BufferState3.WaintingTime := 0;
	                END_IF;

	            END_IF;

	        END_REGION

	        REGION Partially


	            #sR_TRIG_PartialBinReceived(CLK := #sa_TrackingArray_110[#iqUDT_Configuration."110".PEC_EoS.Distance / 10 - 1] <> 0);

	            IF #sR_TRIG_PartialBinReceived.Q THEN

	                IF #iqUDT_PartialBuffer.BufferState1.BinSend AND "DB_GIN".GIN[#sa_TrackingArray_110[#iqUDT_Configuration."110".PEC_EoS.Distance / 10 - 1]].General.Identification.Barcode = #iqUDT_PartialBuffer.BufferState1.UpcomingBarcode THEN

	                    #iqUDT_PartialBuffer.BufferState1 := #iqUDT_PartialBuffer.BufferState2;
	                    #iqUDT_PartialBuffer.BufferState2 := #iqUDT_PartialBuffer.BufferState3;

	                    #iqUDT_PartialBuffer.BufferState3.BinSend := FALSE;
	                    #iqUDT_PartialBuffer.BufferState3.BinRequest := FALSE;
	                    #iqUDT_PartialBuffer.BufferState3.UpcomingBarcode := '';
	                    #iqUDT_PartialBuffer.BufferState3.WaintingTime := 0;
	                END_IF;


	                IF #iqUDT_PartialBuffer.BufferState2.BinSend AND "DB_GIN".GIN[#sa_TrackingArray_110[#iqUDT_Configuration."110".PEC_EoS.Distance / 10 - 1]].General.Identification.Barcode = #iqUDT_PartialBuffer.BufferState2.UpcomingBarcode THEN

	                    #iqUDT_PartialBuffer.BufferState2 := #iqUDT_PartialBuffer.BufferState3;

	                    #iqUDT_PartialBuffer.BufferState3.BinSend := FALSE;
	                    #iqUDT_PartialBuffer.BufferState3.BinRequest := FALSE;
	                    #iqUDT_PartialBuffer.BufferState3.UpcomingBarcode := '';
	                    #iqUDT_PartialBuffer.BufferState3.WaintingTime := 0;
	                END_IF;


	                IF #iqUDT_PartialBuffer.BufferState3.BinSend AND "DB_GIN".GIN[#sa_TrackingArray_110[#iqUDT_Configuration."110".PEC_EoS.Distance / 10 - 1]].General.Identification.Barcode = #iqUDT_PartialBuffer.BufferState3.UpcomingBarcode THEN

	                    #iqUDT_PartialBuffer.BufferState3.BinSend := FALSE;
	                    #iqUDT_PartialBuffer.BufferState3.BinRequest := FALSE;
	                    #iqUDT_PartialBuffer.BufferState3.UpcomingBarcode := '';
	                    #iqUDT_PartialBuffer.BufferState3.WaintingTime := 0;
	                END_IF;

	            END_IF;

	        END_REGION


	    END_REGION
	    *)

	END_REGION

	REGION 010

	    REGION Change GIN range

	        #sR_TRIG_NewParcel010(CLK := #iqUDT_HandshakeUpstream010.GIN <> 0);

	        IF #sR_TRIG_NewParcel010.Q THEN

	            #si_LastGIN010 += 1;

	            IF #si_LastGIN010 < #iqUDT_Configuration.GlobalConfig.GINRangeStart
	                OR #si_LastGIN010 > ((#iqUDT_Configuration.GlobalConfig.GINRangeStart + #iqUDT_Configuration.GlobalConfig.GINRangeEnd) / 2)
	            THEN
	                #si_LastGIN010 := #iqUDT_Configuration.GlobalConfig.GINRangeStart;
	            END_IF;
	            "DB_GIN".GIN[#si_LastGIN010] := "DB_GIN".GIN[#iqUDT_HandshakeUpstream010.GIN];
	            //     #ts_Barcode := "DB_GIN".GIN[#iqUDT_HandshakeUpstream010.GIN].General.Identification.Barcode;
	            //     #ti_DivertDestination := "DB_GIN".GIN[#iqUDT_HandshakeUpstream010.GIN].General.SortStatus.DivertDestination;
	            #iqUDT_HandshakeUpstream010.GIN := #si_LastGIN010;

	            IF "DB_GIN".GIN[#iqUDT_HandshakeUpstream010.GIN].General.SortStatus.GoodDivert
	            THEN
	                "DB_GIN".GIN[#iqUDT_HandshakeUpstream010.GIN].WCS.ReasonCode := '1';
	            ELSE
	                "DB_GIN".GIN[#iqUDT_HandshakeUpstream010.GIN].WCS.ReasonCode := '17';
	            END_IF;


	            //     "DB_GIN".GIN[#iqUDT_HandshakeUpstream010.GIN] := "DB_GINDefault".GIN[#iqUDT_Configuration."010".PEC_EoS.DefaultGIN];
	            //     "DB_GIN".GIN[#iqUDT_HandshakeUpstream010.GIN].General.Identification.Barcode := #ts_Barcode;
	            //     "DB_GIN".GIN[#iqUDT_HandshakeUpstream010.GIN].General.SortStatus.DivertDestination := #ti_DivertDestination;

	            //     "DB_GIN".GIN[#iqUDT_HandshakeUpstream010.GIN].WCS.ReasonCode := '01';

	        END_IF;
	        IF #iqUDT_HandshakeUpstream010.GIN <> 0 THEN
	            #iqUDT_HandshakeUpstream010.GIN := #si_LastGIN010;
	        END_IF;


	    END_REGION

	    REGION Displacement
	        #sFB_Displacement010(#sUDT_Interface_010);
	    END_REGION

	    REGION Tracking

	        #sFB_Tracking_010(iUDT_ConveyorCommonConfiguration := #iqUDT_Configuration."010".Conveyor.Common,
	                          iqa_TrackingData                 := #sa_TrackingArray_010,
	                          iqUDT_ConveyorInterface          := #sUDT_Interface_010,
	                          iqUDT_HandshakeUp                := #iqUDT_HandshakeUpstream010,
	                          iqUDT_Handshake                  := #sUDT_Handshake_010);

	    END_REGION

	    REGION EoS

	        #sFB_PECUpdate_010(iUDT_PECUpdateConfiguration      := #iqUDT_Configuration."010".PEC_EoS,
	                           iUDT_ConveyorCommonConfiguration := #iqUDT_Configuration."010".Conveyor.Common,
	                           ix_PEC                           := #iUDT_MotorInput010.AllSensorPortInputs.LeftSensor,
	                           ix_TeachingMode                  := FALSE,
	                           qUDT_Status                      => #iqUDT_WorkstationStatus."010".PEC_EoS,
	                           iqUDT_ConveyorInterface          := #sUDT_Interface_010,
	                           iqUDT_UnknownGINRange            := #iqUDT_UnknownGINRange,
	                           iqUDT_FifoHeader                 := #sUDT_FifoLostGINHeaderWCS,
	                           iqUDT_Statistics                 := #iqUDT_WorkstationStatistics."010".PEC_EoS,
	                           iqa_TrackingData                 := #sa_TrackingArray_010,
	                           iqa_FifoData                     := #sa_FifoLostGINDataWCS);

	    END_REGION



	    REGION WCS lost in tracking 010
	        "FC_Fifo"(ic_Mode          := 'R',
	                  qUDT_Status      => #tudt_FifoStatus,
	                  qx_Error         => #tx_Dummy,
	                  qx_Warning       => #tx_Dummy,
	                  iqv_Data         := #ti_GIN,
	                  iqUDT_FifoHeader := #sUDT_FifoLostGINHeaderWCS,
	                  iqv_DataBuffer   := #sa_FifoLostGINDataWCS);


	        IF #ti_GIN <> 0 THEN

	            #ta_DestinationArray[1] := #ci_DestinationLeft1;
	            #ta_DestinationArray[2] := #ci_DestinationRight1;
	            #ta_DestinationArray[3] := #ci_DestinationLeft2;
	            #ta_DestinationArray[4] := #ci_DestinationRight2;
	            #ta_DestinationArray[5] := #ci_DestinationStraight;

	            "FC_WCS_ReasonCode"(ii_GIN          := #ti_GIN,
	                                ia_Destinations := #ta_DestinationArray);

	            #sFB_DecisionUpdateWCS_010(is_PLCID            := #iqUDT_Configuration.GlobalConfig.PLCID,
	                                       is_DecisionPoint    := #iqUDT_Configuration.GlobalConfig.WCSDecisionPoint,
	                                       ii_Gin              := #ti_GIN,
	                                       iqUDT_FifoHeader    := #iqUDT_DecisionUpdateHeader,
	                                       iqa_FifoData        := #iqa_DecisionUpdateData,
	                                       iqs_Destinations    := #iqa_DecisionUpdateDestinations,
	                                       iqdi_SequenceNumber := #iqdi_DecisionUpdateSequenceNumber);



	        END_IF;

	    END_REGION


	    REGION WCS Decision update 010

	        #ta_DestinationArray[1] := #ci_DestinationLeft1;
	        #ta_DestinationArray[2] := #ci_DestinationRight1;
	        #ta_DestinationArray[3] := #ci_DestinationLeft2;
	        #ta_DestinationArray[4] := #ci_DestinationRight2;
	        #ta_DestinationArray[5] := #ci_DestinationStraight;


	        "FC_WCS_ReasonCode"(ii_GIN          := #sa_TrackingArray_010[21],
	                            ia_Destinations := #ta_DestinationArray);

	        #sFB_DecisionUpdate_010(is_PLCID            := #iqUDT_Configuration.GlobalConfig.PLCID,
	                                is_DecisionPoint    := #iqUDT_Configuration.GlobalConfig.WCSDecisionPoint,
	                                ii_Gin              := #sa_TrackingArray_010[21],
	                                iqUDT_FifoHeader    := #iqUDT_DecisionUpdateHeader,
	                                iqa_FifoData        := #iqa_DecisionUpdateData,
	                                iqs_Destinations    := #iqa_DecisionUpdateDestinations,
	                                iqdi_SequenceNumber := #iqdi_DecisionUpdateSequenceNumber);



	    END_REGION


	    REGION Conveyor

	        #sFB_Conveyor_010(iUDT_ConveyorConfiguration := #iqUDT_Configuration."010".Conveyor,
	                          idi_PECEoSDistance         := #iqUDT_Configuration."010".PEC_EoS.Distance,
	                          idi_PECBoSDistance         := 0,
	                          ii_ExternalSpeed           := 0,
	                          ix_SafetyOk                := #ix_SafetyOk,
	                          ix_24vOk                   := #ix_24vOk,
	                          ix_400vOk                  := #ix_400vOk,
	                          ix_HardwareOk              := #iUDT_HardwareOk."010",
	                          ix_PECEoS                  := #iqUDT_WorkstationStatus."010".PEC_EoS.PEC,
	                          ix_PECBoS                  := TRUE,
	                          ix_ReverseDirection        := FALSE,
	                          ix_ExternalRequestDieBack  := (#sUDT_Interface_020.ActualSpeed = 0 AND NOT #iqUDT_WorkstationStatus."010".PEC_EoS.PEC),
	                          ix_ExternalRequestHold     := FALSE,
	                          ix_ResetEnergySave         := FALSE,
	                          qUDT_HMIStatus             => #iqUDT_WorkstationStatus."010".Conveyor,
	                          qUDT_Status                => #iqUDT_WorkstationCommonStatus."010",
	                          iqUDT_EquipmentControl     := #iqUDT_EquipmentControl,
	                          iqUDT_ConveyorCommand      := #iqUDT_WorkstationCommands."010".Conveyor,
	                          iqUDT_ConveyorInterface    := #sUDT_Interface_010,
	                          iqUDT_HandShakeUp          := #iqUDT_HandshakeUpstream010,
	                          iqUDT_HandShake            := #sUDT_Handshake_010,
	                          iqUDT_Statistics           := #iqUDT_WorkstationStatistics."010".Conveyor);

	        // #iqUDT_HandshakeUpstream010.RTR := #iqUDT_HandshakeUpstream010.RTR AND #iqUDT_WorkstationStatus."010".PEC_EoS.PEC;

	    END_REGION

	    REGION MCO

	        #sFB_MCOConveyLinxAixController_010(iUDT_AixConfig          := #iqUDT_Configuration."010".MCO_M01,
	                                            iv_AixInputsModule    := #iUDT_MotorInput010,
	                                            ix_24vOk                := #ix_24vOk,
	                                            ix_SimulationModeActive := "DB_Memory".Simulation,
	                                            ii_MotorPositionId      := 1,
	                                            qUDT_HMIStatus          => #iqUDT_WorkstationStatus."010".MCO_M01,
	                                            iqv_AixOutputsModule  := #iqUDT_MotorOutput010,
	                                            iqUDT_ConveyorInterface := #sUDT_Interface_010,
	                                            iqUDT_MCOStatistics     := #iqUDT_WorkstationStatistics."010".MCO_M01);
	    END_REGION

	END_REGION

	REGION 020

	    REGION Displacement
	        #sFB_Displacement020(#sUDT_Interface_020);
	    END_REGION

	    REGION Tracking

	        #sFB_Tracking_020(iUDT_ConveyorCommonConfiguration := #iqUDT_Configuration."020".Conveyor.Common,
	                          iqa_TrackingData                 := #sa_TrackingArray_020,
	                          iqUDT_ConveyorInterface          := #sUDT_Interface_020,
	                          iqUDT_HandshakeUp                := #sUDT_Handshake_010,
	                          iqUDT_Handshake                  := #sUDT_Handshake_020);

	    END_REGION

	    REGION EoS

	        #sFB_PECUpdate_020(iUDT_PECUpdateConfiguration      := #iqUDT_Configuration."020".PEC_EoS,
	                           iUDT_ConveyorCommonConfiguration := #iqUDT_Configuration."020".Conveyor.Common,
	                           ix_PEC                           := #iUDT_MotorInput010.AllSensorPortInputs.RightSensor,
	                           ix_TeachingMode                  := FALSE,
	                           qUDT_Status                      => #iqUDT_WorkstationStatus."020".PEC_EoS,
	                           iqUDT_ConveyorInterface          := #sUDT_Interface_020,
	                           iqUDT_UnknownGINRange            := #iqUDT_UnknownGINRange,
	                           iqUDT_FifoHeader                 := #sUDT_FifoLostGINHeader,
	                           iqUDT_Statistics                 := #iqUDT_WorkstationStatistics."020".PEC_EoS,
	                           iqa_TrackingData                 := #sa_TrackingArray_020,
	                           iqa_FifoData                     := #sa_FifoLostGINData);




	    END_REGION

	    REGION Conveyor

	        #sFB_Conveyor_020(iUDT_ConveyorConfiguration := #iqUDT_Configuration."020".Conveyor,
	                          idi_PECEoSDistance         := #iqUDT_Configuration."020".PEC_EoS.Distance,
	                          idi_PECBoSDistance         := 0,
	                          ii_ExternalSpeed           := 0,
	                          ix_SafetyOk                := #ix_SafetyOk,
	                          ix_24vOk                   := #ix_24vOk,
	                          ix_400vOk                  := #ix_400vOk,
	                          ix_HardwareOk              := #iUDT_HardwareOk."010",
	                          ix_PECEoS                  := #iqUDT_WorkstationStatus."020".PEC_EoS.PEC,
	                          ix_PECBoS                  := TRUE,
	                          ix_ReverseDirection        := FALSE,
	                          ix_ExternalRequestDieBack  := #sx_Hold020 OR (#sUDT_Interface_030.ActualSpeed = 0 AND NOT #iqUDT_WorkstationStatus."020".PEC_EoS.PEC),
	                          ix_ExternalRequestHold     := FALSE,
	                          ix_ResetEnergySave         := FALSE,
	                          qUDT_HMIStatus             => #iqUDT_WorkstationStatus."020".Conveyor,
	                          qUDT_Status                => #iqUDT_WorkstationCommonStatus."020",
	                          iqUDT_EquipmentControl     := #iqUDT_EquipmentControl,
	                          iqUDT_ConveyorCommand      := #iqUDT_WorkstationCommands."020".Conveyor,
	                          iqUDT_ConveyorInterface    := #sUDT_Interface_020,
	                          iqUDT_HandShakeUp          := #sUDT_Handshake_010,
	                          iqUDT_HandShake            := #sUDT_Handshake_020,
	                          iqUDT_Statistics           := #iqUDT_WorkstationStatistics."020".Conveyor);

	    END_REGION

	    REGION MCO

	        #sFB_MCOConveyLinxAixController_020(iUDT_AixConfig          := #iqUDT_Configuration."020".MCO_M01,
	                                            iv_AixInputsModule    := #iUDT_MotorInput010,
	                                            ix_24vOk                := #ix_24vOk,
	                                            ix_SimulationModeActive := "DB_Memory".Simulation,
	                                            ii_MotorPositionId      := 2,
	                                            qUDT_HMIStatus          => #iqUDT_WorkstationStatus."020".MCO_M01,
	                                            iqv_AixOutputsModule  := #iqUDT_MotorOutput010,
	                                            iqUDT_ConveyorInterface := #sUDT_Interface_020,
	                                            iqUDT_MCOStatistics     := #iqUDT_WorkstationStatistics."020".MCO_M01);
	    END_REGION

	END_REGION

	REGION 030

	    REGION Displacement
	        #sFB_Displacement030(#sUDT_Interface_030);
	    END_REGION

	    REGION Tracking

	        #sFB_Tracking_030(iUDT_ConveyorCommonConfiguration := #iqUDT_Configuration."030".Conveyor.Common,
	                          iqa_TrackingData                 := #sa_TrackingArray_030,
	                          iqUDT_ConveyorInterface          := #sUDT_Interface_030,
	                          iqUDT_HandshakeUp                := #sUDT_Handshake_020,
	                          iqUDT_Handshake                  := #sUDT_Handshake_030);

	    END_REGION

	    REGION EoS

	        #sFB_PECUpdate_030(iUDT_PECUpdateConfiguration      := #iqUDT_Configuration."030".PEC_EoS,
	                           iUDT_ConveyorCommonConfiguration := #iqUDT_Configuration."030".Conveyor.Common,
	                           ix_PEC                           := #iUDT_MotorInput030.AllSensorPortInputs.LeftSensor,
	                           ix_TeachingMode                  := FALSE,
	                           qUDT_Status                      => #iqUDT_WorkstationStatus."030".PEC_EoS,
	                           iqUDT_ConveyorInterface          := #sUDT_Interface_030,
	                           iqUDT_UnknownGINRange            := #iqUDT_UnknownGINRange,
	                           iqUDT_FifoHeader                 := #sUDT_FifoLostGINHeader,
	                           iqUDT_Statistics                 := #iqUDT_WorkstationStatistics."030".PEC_EoS,
	                           iqa_TrackingData                 := #sa_TrackingArray_030,
	                           iqa_FifoData                     := #sa_FifoLostGINData);




	    END_REGION

	    REGION Conveyor

	        #sUDT_Handshake_030.RTR := #sUDT_Handshake_030.RTR AND NOT #sx_Hold030 OR #iqUDT_WorkstationStatus."030".PEC_EoS.PEC;


	        #sFB_Conveyor_030(iUDT_ConveyorConfiguration := #iqUDT_Configuration."030".Conveyor,
	                          idi_PECEoSDistance         := #iqUDT_Configuration."030".PEC_EoS.Distance,
	                          idi_PECBoSDistance         := 0,
	                          ii_ExternalSpeed           := 0,
	                          ix_SafetyOk                := #ix_SafetyOk,
	                          ix_24vOk                   := #ix_24vOk,
	                          ix_400vOk                  := #ix_400vOk,
	                          ix_HardwareOk              := #iUDT_HardwareOk."030",
	                          ix_PECEoS                  := #iqUDT_WorkstationStatus."030".PEC_EoS.PEC,
	                          ix_PECBoS                  := TRUE,
	                          ix_ReverseDirection        := FALSE,
	                          ix_ExternalRequestDieBack  := FALSE,
	                          ix_ExternalRequestHold     := #sx_Hold030,
	                          ix_ResetEnergySave         := FALSE,
	                          qUDT_HMIStatus             => #iqUDT_WorkstationStatus."030".Conveyor,
	                          qUDT_Status                => #iqUDT_WorkstationCommonStatus."030",
	                          iqUDT_EquipmentControl     := #iqUDT_EquipmentControl,
	                          iqUDT_ConveyorCommand      := #iqUDT_WorkstationCommands."030".Conveyor,
	                          iqUDT_ConveyorInterface    := #sUDT_Interface_030,
	                          iqUDT_HandShakeUp          := #sUDT_Handshake_020,
	                          iqUDT_HandShake            := #sUDT_Handshake_030,
	                          iqUDT_Statistics           := #iqUDT_WorkstationStatistics."030".Conveyor);

	    END_REGION

	    REGION MCO

	        #sFB_MCOConveyLinxAixController_030(iUDT_AixConfig          := #iqUDT_Configuration."030".MCO_M01,
	                                            iv_AixInputsModule    := #iUDT_MotorInput030,
	                                            ix_24vOk                := #ix_24vOk,
	                                            ix_SimulationModeActive := "DB_Memory".Simulation,
	                                            ii_MotorPositionId      := 1,
	                                            qUDT_HMIStatus          => #iqUDT_WorkstationStatus."030".MCO_M01,
	                                            iqv_AixOutputsModule  := #iqUDT_MotorOutput030,
	                                            iqUDT_ConveyorInterface := #sUDT_Interface_030,
	                                            iqUDT_MCOStatistics     := #iqUDT_WorkstationStatistics."030".MCO_M01);
	    END_REGION

	END_REGION

	REGION 040

	    REGION Displacement
	        #sFB_Displacement040(#sUDT_Interface_040);
	    END_REGION

	    REGION MCO

	        #sFB_MCOConveyLinxAixController_040(iUDT_AixConfig          := #iqUDT_Configuration."040".MCO_M01,
	                                            iv_AixInputsModule    := #iUDT_MotorInput040,
	                                            ii_PositionSetpoint     := #iqUDT_RATPositioning040.Lower.EndPosition,
	                                            ix_24vOk                := #ix_24vOk,
	                                            ix_SimulationModeActive := "DB_Memory".Simulation,
	                                            ii_MotorPositionId      := 1,
	                                            ix_StartPositioning     := #iqUDT_RATPositioning040.Lower.Start,
	                                            ix_ResetPosition        := #iqUDT_RATPositioning040.Lower.ResetPosition,
	                                            qUDT_HMIStatus          => #iqUDT_WorkstationStatus."040".MCO_M01,
	                                            qx_Positioned           => #iqUDT_RATPositioning040.Lower.Done,
	                                            iqv_AixOutputsModule  := #iqUDT_MotorOutput040,
	                                            iqUDT_ConveyorInterface := #sUDT_Interface_040,
	                                            iqUDT_MCOStatistics     := #iqUDT_WorkstationStatistics."040".MCO_M01);
	    END_REGION

	    REGION BladeStopEoS

	        IF #iqUDT_Configuration.GlobalConfig.StationVariant = 1 OR #iqUDT_Configuration.GlobalConfig.StationVariant = 2 OR #iqUDT_Configuration.GlobalConfig.StationVariant = 5 OR #iqUDT_Configuration.GlobalConfig.StationVariant = 6 THEN

	            #sFB_BladeStopEoS_040(iUDT_Configuration     := #iqUDT_Configuration."040".BladeStopEoS,
	                                  ix_IsOpened            := #ix_BladeStopIsUp040,
	                                  ix_IsClosed            := #ix_BladeStopIsDown040,
	                                  ix_AirPressureOk       := TRUE,
	                                  qx_Open                => #qx_BladeStopControl040,
	                                  qUDT_HMIStatus         => #iqUDT_WorkstationStatus."040".BladeStopEoS,
	                                  iqUDT_Statistics       := #iqUDT_WorkstationStatistics."040".BladeStopEoS,
	                                  iqUDT_EquipmentControl := #iqUDT_EquipmentControl,
	                                  iqUDT_HMICommand       := #iqUDT_WorkstationCommands."040".BladeStopEoS,
	                                  iqUDT_Interface        := #sUDT_Interface_040_BladeStopEoS);
	        END_IF;

	    END_REGION

	END_REGION

	REGION 041

	    REGION Displacement
	        #sFB_Displacement041(#sUDT_Interface_041);
	    END_REGION

	    REGION RAT

	        // #iqUDT_Configuration."041".RightAngledTransfer.BladeStop := #iqUDT_Configuration.GlobalConfig.StationVariant = 1
	        // OR #iqUDT_Configuration.GlobalConfig.StationVariant = 2
	        // OR #iqUDT_Configuration.GlobalConfig.StationVariant = 5
	        // OR #iqUDT_Configuration.GlobalConfig.StationVariant = 6;

	        IF #iqUDT_Configuration.GlobalConfig.StationVariant = 1 OR #iqUDT_Configuration.GlobalConfig.StationVariant = 3 OR #iqUDT_Configuration.GlobalConfig.StationVariant = 5 THEN
	            #sUDT_Handshake_041C := #sUDT_Handshake_241C;
	        ELSIF #iqUDT_Configuration.GlobalConfig.StationVariant = 2 OR #iqUDT_Configuration.GlobalConfig.StationVariant = 4 OR #iqUDT_Configuration.GlobalConfig.StationVariant = 6 THEN
	            #sUDT_Handshake_041D := #sUDT_Handshake_241D;
	        END_IF;


	        #sFB_RightAngledTransfer_041(iUDT_Configuration              := #iqUDT_Configuration."041".RightAngledTransfer,
	                                     iUDT_LowerConveyorConfiguration := #iqUDT_Configuration."040".Conveyor,
	                                     iUDT_UpperConveyorConfiguration := #iqUDT_Configuration."041".Conveyor,
	                                     iUDT_PECConfiguration           := #iqUDT_Configuration."040".PEC_EoS,
	                                     ii_DestinationA                 := #si_040DestinationA,
	                                     ii_DestinationB                 := #si_040DestinationB,
	                                     ii_DestinationC                 := #si_040DestinationC,
	                                     ii_DestinationD                 := #si_040DestinationD,
	                                     ix_HardwareOk                   := #iUDT_HardwareOk."040",
	                                     ix_400vOk                       := #ix_400vOk,
	                                     ix_24vOk                        := #ix_24vOk,
	                                     ix_SafetyOk                     := #ix_SafetyOk,
	                                     ix_AirPressureOk                := #ix_AirPressureOk,
	                                     ix_SectionIsDown                := #ix_SectionIsDown041,
	                                     ix_SectionIsUp                  := #ix_SectionIsUp041,
	                                     ix_ConveyorAAuto                := #iqUDT_WorkstationCommonStatus."030".AutoON,
	                                     ix_ConveyorBAuto                := #iqUDT_WorkstationCommonStatus."050".AutoON,
	                                     ix_ConveyorCAuto                := #iqUDT_WorkstationCommonStatus."241".AutoON AND (#iqUDT_Configuration.GlobalConfig.StationVariant = 1 OR #iqUDT_Configuration.GlobalConfig.StationVariant = 3 OR #iqUDT_Configuration.GlobalConfig.StationVariant = 5),
	                                     ix_ConveyorDAuto                := #iqUDT_WorkstationCommonStatus."241".AutoON AND (#iqUDT_Configuration.GlobalConfig.StationVariant = 2 OR #iqUDT_Configuration.GlobalConfig.StationVariant = 4 OR #iqUDT_Configuration.GlobalConfig.StationVariant = 6),
	                                     ix_PEC                          := #iUDT_MotorInput040.AllSensorPortInputs.LeftSensor,
	                                     ix_ExternalReceiveRequestA      := NOT #iqUDT_WorkstationStatus."030".PEC_EoS.PEC AND #sx_Enable0X0In,
	                                     ix_ExternalReceiveRequestB      := false,
	                                     ix_ExternalReceiveRequestC      := #sFB_RightAngledTransfer_241.qx_ExternalSendRequestC AND (#iqUDT_Configuration.GlobalConfig.StationVariant = 1 OR #iqUDT_Configuration.GlobalConfig.StationVariant = 3 OR #iqUDT_Configuration.GlobalConfig.StationVariant = 5),
	                                     ix_ExternalReceiveRequestD      := #sFB_RightAngledTransfer_241.qx_ExternalSendRequestD AND (#iqUDT_Configuration.GlobalConfig.StationVariant = 2 OR #iqUDT_Configuration.GlobalConfig.StationVariant = 4 OR #iqUDT_Configuration.GlobalConfig.StationVariant = 6),
	                                     ix_PECInfeedA                   := #iqUDT_WorkstationStatus."030".PEC_EoS.PEC,
	                                     ix_PECInfeedC                   := #iqUDT_WorkstationStatus."240".PEC_EoS.PEC AND (#iqUDT_Configuration.GlobalConfig.StationVariant = 1 OR #iqUDT_Configuration.GlobalConfig.StationVariant = 3 OR #iqUDT_Configuration.GlobalConfig.StationVariant = 5),
	                                     ix_PECInfeedD                   := #iqUDT_WorkstationStatus."240".PEC_EoS.PEC AND (#iqUDT_Configuration.GlobalConfig.StationVariant = 2 OR #iqUDT_Configuration.GlobalConfig.StationVariant = 4 OR #iqUDT_Configuration.GlobalConfig.StationVariant = 6),
	                                     qUDT_HMIRATStatus               => #iqUDT_WorkstationStatus."041".RightAngledTransfer,
	                                     qUDT_HMIConveyorStatus          => #iqUDT_WorkstationStatus."040".Conveyor,
	                                     qUDT_HMIPECStatus               => #iqUDT_WorkstationStatus."040".PEC_EoS,
	                                     qUDT_RATStatus                  => #iqUDT_WorkstationCommonStatus."041",
	                                     qUDT_ConveyorStatus             => #iqUDT_WorkstationCommonStatus."040",
	                                     qx_PopupControl                 => #qx_PopupControl041,
	                                     iqUDT_EquipmentControl          := #iqUDT_EquipmentControl,
	                                     iqUDT_RATCommand                := #iqUDT_WorkstationCommands."041".RightAngledTransfer,
	                                     iqUDT_ConveyorCommand           := #iqUDT_WorkstationCommands."040".Conveyor,
	                                     iqUDT_RATStatistics             := #iqUDT_WorkstationStatistics."041".RightAngledTransfer,
	                                     iqUDT_ConveyorStatistics        := #iqUDT_WorkstationStatistics."040".Conveyor,
	                                     iqUDT_PECStatistics             := #iqUDT_WorkstationStatistics."040".PEC_EoS,
	                                     iqUDT_HandShakeConveyorA        := #sUDT_Handshake_030,
	                                     iqUDT_HandShakeConveyorB        := #sUDT_Handshake_040,
	                                     iqUDT_HandShakeConveyorC        := #sUDT_Handshake_041C,
	                                     iqUDT_HandShakeConveyorD        := #sUDT_Handshake_041D,
	                                     iqUDT_LowerConveyorInterface    := #sUDT_Interface_040,
	                                     iqUDT_UpperConveyorInterface    := #sUDT_Interface_041,
	                                     iqUDT_RATPositioning            := #iqUDT_RATPositioning040,
	                                     iqUDT_BladeStopEoSInterface     := #sUDT_Interface_040_BladeStopEoS,
	                                     iqUDT_BladeStopBoSInterface     := #tUDT_DummyBladeStop);

	    END_REGION

	    IF #iqUDT_Configuration.GlobalConfig.StationVariant = 1 OR #iqUDT_Configuration.GlobalConfig.StationVariant = 3 OR #iqUDT_Configuration.GlobalConfig.StationVariant = 5 THEN
	        #sUDT_Handshake_241C := #sUDT_Handshake_041C;
	    ELSIF #iqUDT_Configuration.GlobalConfig.StationVariant = 2 OR #iqUDT_Configuration.GlobalConfig.StationVariant = 4 OR #iqUDT_Configuration.GlobalConfig.StationVariant = 6 THEN
	        #sUDT_Handshake_241D := #sUDT_Handshake_041D;
	    END_IF;



	    REGION MCO

	        #sFB_MCOConveyLinxAixController_041(iUDT_AixConfig          := #iqUDT_Configuration."041".MCO_M01,
	                                            iv_AixInputsModule    := #iUDT_MotorInput040,
	                                            ii_PositionSetpoint     := #iqUDT_RATPositioning040.Upper.EndPosition,
	                                            ix_24vOk                := #ix_24vOk,
	                                            ix_SimulationModeActive := "DB_Memory".Simulation,
	                                            ii_MotorPositionId      := 2,
	                                            ix_StartPositioning     := #iqUDT_RATPositioning040.Upper.Start,
	                                            qUDT_HMIStatus          => #iqUDT_WorkstationStatus."041".MCO_M01,
	                                            qx_Positioned           => #iqUDT_RATPositioning040.Upper.Done,
	                                            iqv_AixOutputsModule  := #iqUDT_MotorOutput040,
	                                            iqUDT_ConveyorInterface := #sUDT_Interface_041,
	                                            iqUDT_MCOStatistics     := #iqUDT_WorkstationStatistics."041".MCO_M01);
	    END_REGION

	END_REGION

	IF #iqUDT_Configuration.GlobalConfig.StationVariant = 1 OR #iqUDT_Configuration.GlobalConfig.StationVariant = 2 OR #iqUDT_Configuration.GlobalConfig.StationVariant = 5 OR #iqUDT_Configuration.GlobalConfig.StationVariant = 6 THEN

	    REGION 050

	        REGION Displacement
	            #sFB_Displacement050(#sUDT_Interface_050);
	        END_REGION

	        REGION Tracking

	            #sFB_Tracking_050(iUDT_ConveyorCommonConfiguration := #iqUDT_Configuration."050".Conveyor.Common,
	                              iqa_TrackingData                 := #sa_TrackingArray_050,
	                              iqUDT_ConveyorInterface          := #sUDT_Interface_050,
	                              iqUDT_HandshakeUp                := #sUDT_Handshake_040,
	                              iqUDT_Handshake                  := #sUDT_Handshake_050);

	        END_REGION

	        REGION EoS

	            #sFB_PECUpdate_050(iUDT_PECUpdateConfiguration      := #iqUDT_Configuration."050".PEC_EoS,
	                               iUDT_ConveyorCommonConfiguration := #iqUDT_Configuration."050".Conveyor.Common,
	                               ix_PEC                           := NOT #iUDT_MotorInput050.AllSensorPortInputs.LeftSensor,
	                               ix_TeachingMode                  := FALSE,
	                               qUDT_Status                      => #iqUDT_WorkstationStatus."050".PEC_EoS,
	                               iqUDT_ConveyorInterface          := #sUDT_Interface_050,
	                               iqUDT_UnknownGINRange            := #iqUDT_UnknownGINRange,
	                               iqUDT_FifoHeader                 := #sUDT_FifoLostGINHeader,
	                               iqUDT_Statistics                 := #iqUDT_WorkstationStatistics."050".PEC_EoS,
	                               iqa_TrackingData                 := #sa_TrackingArray_050,
	                               iqa_FifoData                     := #sa_FifoLostGINData);

	        END_REGION

	        REGION Conveyor

	            //#sUDT_Handshake_050.RTR := TRUE;

	            #sUDT_Handshake_050.RTR := (#iqUDT_WorkstationStatus."060".PEC_EoS.PEC AND #sUDT_Interface_060.ActualSpeed <> 0)
	            OR (#iqUDT_WorkstationStatus."050".PEC_EoS.PEC);

	            #sFB_Conveyor_050(iUDT_ConveyorConfiguration := #iqUDT_Configuration."050".Conveyor,
	                              idi_PECEoSDistance         := #iqUDT_Configuration."050".PEC_EoS.Distance,
	                              idi_PECBoSDistance         := 0,
	                              ii_ExternalSpeed           := 0,
	                              ix_SafetyOk                := #ix_SafetyOk,
	                              ix_24vOk                   := #ix_24vOk,
	                              ix_400vOk                  := #ix_400vOk,
	                              ix_HardwareOk              := #iUDT_HardwareOk."050",
	                              ix_PECEoS                  := #iqUDT_WorkstationStatus."050".PEC_EoS.PEC,
	                              ix_PECBoS                  := TRUE,
	                              ix_ReverseDirection        := FALSE,
	                              ix_ExternalRequestDieBack  := FALSE,
	                              ix_ExternalRequestHold     := #sx_ReleaseBinHold0X0,//sx_Hold050,//NOT #tx_Enable,
	                              ix_ResetEnergySave         := FALSE,
	                              qUDT_HMIStatus             => #iqUDT_WorkstationStatus."050".Conveyor,
	                              qUDT_Status                => #iqUDT_WorkstationCommonStatus."050",
	                              iqUDT_EquipmentControl     := #iqUDT_EquipmentControl,
	                              iqUDT_ConveyorCommand      := #iqUDT_WorkstationCommands."050".Conveyor,
	                              iqUDT_ConveyorInterface    := #sUDT_Interface_050,
	                              iqUDT_HandShakeUp          := #sUDT_Handshake_040,
	                              iqUDT_HandShake            := #sUDT_Handshake_050,
	                              iqUDT_Statistics           := #iqUDT_WorkstationStatistics."050".Conveyor);

	        END_REGION



	        REGION MCO

	            #sFB_MCOConveyLinxAixController_050(iUDT_AixConfig          := #iqUDT_Configuration."050".MCO_M01,
	                                                iv_AixInputsModule    := #iUDT_MotorInput050,
	                                                ix_24vOk                := #ix_24vOk,
	                                                ix_SimulationModeActive := "DB_Memory".Simulation,
	                                                ii_MotorPositionId      := 1,
	                                                qUDT_HMIStatus          => #iqUDT_WorkstationStatus."050".MCO_M01,
	                                                iqv_AixOutputsModule  := #iqUDT_MotorOutput050,
	                                                iqUDT_ConveyorInterface := #sUDT_Interface_050,
	                                                iqUDT_MCOStatistics     := #iqUDT_WorkstationStatistics."050".MCO_M01);
	        END_REGION

	    END_REGION

	    REGION 060

	        REGION Displacement
	            #sFB_Displacement060(#sUDT_Interface_060);
	        END_REGION

	        REGION Tracking

	            #sFB_Tracking_060(iUDT_ConveyorCommonConfiguration := #iqUDT_Configuration."060".Conveyor.Common,
	                              iqa_TrackingData                 := #sa_TrackingArray_060,
	                              iqUDT_ConveyorInterface          := #sUDT_Interface_060,
	                              iqUDT_HandshakeUp                := #sUDT_Handshake_050,
	                              iqUDT_Handshake                  := #sUDT_Handshake_060);

	        END_REGION

	        REGION EoS

	            #sFB_PECUpdate_060(iUDT_PECUpdateConfiguration      := #iqUDT_Configuration."060".PEC_EoS,
	                               iUDT_ConveyorCommonConfiguration := #iqUDT_Configuration."060".Conveyor.Common,
	                               ix_PEC                           := NOT #iUDT_MotorInput050.AllSensorPortInputs.RightSensor,
	                               ix_TeachingMode                  := FALSE,
	                               qUDT_Status                      => #iqUDT_WorkstationStatus."060".PEC_EoS,
	                               iqUDT_ConveyorInterface          := #sUDT_Interface_060,
	                               iqUDT_UnknownGINRange            := #iqUDT_UnknownGINRange,
	                               iqUDT_FifoHeader                 := #sUDT_FifoLostGINHeader,
	                               iqUDT_Statistics                 := #iqUDT_WorkstationStatistics."060".PEC_EoS,
	                               iqa_TrackingData                 := #sa_TrackingArray_060,
	                               iqa_FifoData                     := #sa_FifoLostGINData);

	        END_REGION

	        REGION Conveyor

	            // #sUDT_Handshake_060.RTR := TRUE;

	            #sUDT_Handshake_060.RTR := (#iqUDT_WorkstationStatus."070".PEC_EoS.PEC AND #sUDT_Interface_070.ActualSpeed <> 0)
	            OR (#iqUDT_WorkstationStatus."060".PEC_EoS.PEC);

	            #sFB_Conveyor_060(iUDT_ConveyorConfiguration := #iqUDT_Configuration."060".Conveyor,
	                              idi_PECEoSDistance         := #iqUDT_Configuration."060".PEC_EoS.Distance,
	                              idi_PECBoSDistance         := 0,
	                              ii_ExternalSpeed           := 0,
	                              ix_SafetyOk                := #ix_SafetyOk,
	                              ix_24vOk                   := #ix_24vOk,
	                              ix_400vOk                  := #ix_400vOk,
	                              ix_HardwareOk              := #iUDT_HardwareOk."050",
	                              ix_PECEoS                  := #iqUDT_WorkstationStatus."060".PEC_EoS.PEC,
	                              ix_PECBoS                  := TRUE,
	                              ix_ReverseDirection        := FALSE,
	                              ix_ExternalRequestDieBack  := FALSE,
	                              ix_ExternalRequestHold     := #sx_Hold060,//NOT #tx_Enable,//(NOT #iqUDT_WorkstationStatus."035"."036".PEC_EoS.PEC AND NOT #iqUDT_WorkstationStatus."030"."031".PEC_EoS.PEC) OR (#sUDT_Interface_036.ActualSpeed = 0 AND #iqUDT_WorkstationStatus."030"."031".PEC_EoS.PEC),
	                              ix_ResetEnergySave         := FALSE,
	                              qUDT_HMIStatus             => #iqUDT_WorkstationStatus."060".Conveyor,
	                              qUDT_Status                => #iqUDT_WorkstationCommonStatus."060",
	                              iqUDT_EquipmentControl     := #iqUDT_EquipmentControl,
	                              iqUDT_ConveyorCommand      := #iqUDT_WorkstationCommands."060".Conveyor,
	                              iqUDT_ConveyorInterface    := #sUDT_Interface_060,
	                              iqUDT_HandShakeUp          := #sUDT_Handshake_050,
	                              iqUDT_HandShake            := #sUDT_Handshake_060,
	                              iqUDT_Statistics           := #iqUDT_WorkstationStatistics."060".Conveyor);

	        END_REGION

	        REGION MCO

	            #sFB_MCOConveyLinxAixController_060(iUDT_AixConfig          := #iqUDT_Configuration."060".MCO_M01,
	                                                iv_AixInputsModule    := #iUDT_MotorInput050,
	                                                ix_24vOk                := #ix_24vOk,
	                                                ix_SimulationModeActive := "DB_Memory".Simulation,
	                                                ii_MotorPositionId      := 2,
	                                                qUDT_HMIStatus          => #iqUDT_WorkstationStatus."060".MCO_M01,
	                                                iqv_AixOutputsModule  := #iqUDT_MotorOutput050,
	                                                iqUDT_ConveyorInterface := #sUDT_Interface_060,
	                                                iqUDT_MCOStatistics     := #iqUDT_WorkstationStatistics."060".MCO_M01);
	        END_REGION

	    END_REGION

	    REGION 070

	        REGION Displacement
	            #sFB_Displacement070(#sUDT_Interface_070);
	        END_REGION

	        REGION Tracking

	            #sFB_Tracking_070(iUDT_ConveyorCommonConfiguration := #iqUDT_Configuration."070".Conveyor.Common,
	                              iqa_TrackingData                 := #sa_TrackingArray_070,
	                              iqUDT_ConveyorInterface          := #sUDT_Interface_070,
	                              iqUDT_HandshakeUp                := #sUDT_Handshake_060,
	                              iqUDT_Handshake                  := #sUDT_Handshake_070);

	        END_REGION

	        REGION EoS

	            #sFB_PECUpdate_070(iUDT_PECUpdateConfiguration      := #iqUDT_Configuration."070".PEC_EoS,
	                               iUDT_ConveyorCommonConfiguration := #iqUDT_Configuration."070".Conveyor.Common,
	                               ix_PEC                           := NOT #iUDT_MotorInput070.AllSensorPortInputs.LeftSensor,
	                               ix_TeachingMode                  := FALSE,
	                               qUDT_Status                      => #iqUDT_WorkstationStatus."070".PEC_EoS,
	                               iqUDT_ConveyorInterface          := #sUDT_Interface_070,
	                               iqUDT_UnknownGINRange            := #iqUDT_UnknownGINRange,
	                               iqUDT_FifoHeader                 := #sUDT_FifoLostGINHeader,
	                               iqUDT_Statistics                 := #iqUDT_WorkstationStatistics."070".PEC_EoS,
	                               iqa_TrackingData                 := #sa_TrackingArray_070,
	                               iqa_FifoData                     := #sa_FifoLostGINData);

	        END_REGION

	        REGION Conveyor

	            #sUDT_Handshake_070.RTR := #iqUDT_WorkstationStatus."070".PEC_EoS.PEC;

	            #sFB_Conveyor_070(iUDT_ConveyorConfiguration := #iqUDT_Configuration."070".Conveyor,
	                              idi_PECEoSDistance         := #iqUDT_Configuration."070".PEC_EoS.Distance,
	                              idi_PECBoSDistance         := 0,
	                              ii_ExternalSpeed           := 0,
	                              ix_SafetyOk                := #ix_SafetyOk,
	                              ix_24vOk                   := #ix_24vOk,
	                              ix_400vOk                  := #ix_400vOk,
	                              ix_HardwareOk              := #iUDT_HardwareOk."070",
	                              ix_PECEoS                  := #iqUDT_WorkstationStatus."070".PEC_EoS.PEC,
	                              ix_PECBoS                  := TRUE,
	                              ix_ReverseDirection        := FALSE,
	                              ix_ExternalRequestDieBack  := FALSE,
	                              ix_ExternalRequestHold     := #sx_Hold070,
	                              ix_ResetEnergySave         := FALSE,
	                              qUDT_HMIStatus             => #iqUDT_WorkstationStatus."070".Conveyor,
	                              qUDT_Status                => #iqUDT_WorkstationCommonStatus."070",
	                              iqUDT_EquipmentControl     := #iqUDT_EquipmentControl,
	                              iqUDT_ConveyorCommand      := #iqUDT_WorkstationCommands."070".Conveyor,
	                              iqUDT_ConveyorInterface    := #sUDT_Interface_070,
	                              iqUDT_HandShakeUp          := #sUDT_Handshake_060,
	                              iqUDT_HandShake            := #sUDT_Handshake_070,
	                              iqUDT_Statistics           := #iqUDT_WorkstationStatistics."070".Conveyor);

	        END_REGION

	        REGION MCO

	            #sFB_MCOConveyLinxAixController_070(iUDT_AixConfig          := #iqUDT_Configuration."070".MCO_M01,
	                                                iv_AixInputsModule    := #iUDT_MotorInput070,
	                                                ix_24vOk                := #ix_24vOk,
	                                                ix_SimulationModeActive := "DB_Memory".Simulation,
	                                                ii_MotorPositionId      := 1,
	                                                qUDT_HMIStatus          => #iqUDT_WorkstationStatus."070".MCO_M01,
	                                                iqv_AixOutputsModule  := #iqUDT_MotorOutput070,
	                                                iqUDT_ConveyorInterface := #sUDT_Interface_070,
	                                                iqUDT_MCOStatistics     := #iqUDT_WorkstationStatistics."070".MCO_M01);
	        END_REGION

	    END_REGION



	    REGION 080

	        REGION Displacement
	            #sFB_Displacement080(#sUDT_Interface_080);
	        END_REGION
	        (*
	        REGION EoS
	            #sFB_PEC_080(ix_PEC                  := #iUDT_MotorInput070.AllSensorPortInputs.RightSensor,
	                         iUDT_PECConfiguration   := #iqUDT_Configuration."080".PEC_EoS,
	                         qUDT_HMIStatus          => #iqUDT_WorkstationStatus."080".PEC_EoS,
	                         iqUDT_ConveyorInterface := #sUDT_Interface_080,
	                         iqUDT_PECStatistics     := #iqUDT_WorkstationStatistics."080".PEC_EoS);
	        END_REGION
	        *)

	        REGION Conveyor

	            #sUDT_Handshake_080.RTR := TRUE;

	            #sFB_Conveyor_080(iUDT_ConveyorConfiguration := #iqUDT_Configuration."080".Conveyor,
	                              idi_PECEoSDistance         := 0,
	                              idi_PECBoSDistance         := 0,
	                              ii_ExternalSpeed           := 0,
	                              ix_SafetyOk                := #ix_SafetyOk,
	                              ix_24vOk                   := #ix_24vOk,
	                              ix_400vOk                  := #ix_400vOk,
	                              ix_HardwareOk              := #iUDT_HardwareOk."070",
	                              ix_PECEoS                  := TRUE,
	                              ix_PECBoS                  := TRUE,
	                              ix_ReverseDirection        := FALSE,
	                              ix_ExternalRequestDieBack  := FALSE,
	                              ix_ExternalRequestHold     := #sx_Hold080,
	                              ix_ResetEnergySave         := NOT #sx_Hold080,
	                              qUDT_HMIStatus             => #iqUDT_WorkstationStatus."080".Conveyor,
	                              qUDT_Status                => #iqUDT_WorkstationCommonStatus."080",
	                              iqUDT_EquipmentControl     := #iqUDT_EquipmentControl,
	                              iqUDT_ConveyorCommand      := #iqUDT_WorkstationCommands."080".Conveyor,
	                              iqUDT_ConveyorInterface    := #sUDT_Interface_080,
	                              iqUDT_HandShakeUp          := #sUDT_HandshakeUp_080,
	                              iqUDT_HandShake            := #sUDT_Handshake_080,
	                              iqUDT_Statistics           := #iqUDT_WorkstationStatistics."080".Conveyor);

	        END_REGION

	        REGION MCO

	            #sFB_MCOConveyLinxAixController_080(iUDT_AixConfig          := #iqUDT_Configuration."080".MCO_M01,
	                                                iv_AixInputsModule    := #iUDT_MotorInput070,
	                                                ix_24vOk                := #ix_24vOk,
	                                                ix_SimulationModeActive := "DB_Memory".Simulation,
	                                                ii_MotorPositionId      := 2,
	                                                qUDT_HMIStatus          => #iqUDT_WorkstationStatus."080".MCO_M01,
	                                                iqv_AixOutputsModule  := #iqUDT_MotorOutput070,
	                                                iqUDT_ConveyorInterface := #sUDT_Interface_080,
	                                                iqUDT_MCOStatistics     := #iqUDT_WorkstationStatistics."080".MCO_M01);
	        END_REGION

	    END_REGION
	END_IF;

	REGION 110

	    REGION Change GIN range

	        #sR_TRIG_NewParcel110(CLK := #iqUDT_HandshakeUpstream110.GIN <> 0);

	        IF #sR_TRIG_NewParcel110.Q THEN

	            #si_LastGIN110 += 1;

	            IF #si_LastGIN110 < ((#iqUDT_Configuration.GlobalConfig.GINRangeStart + #iqUDT_Configuration.GlobalConfig.GINRangeEnd) / 2) + 1
	                OR #si_LastGIN110 > #iqUDT_Configuration.GlobalConfig.GINRangeEnd
	            THEN
	                #si_LastGIN110 := ((#iqUDT_Configuration.GlobalConfig.GINRangeStart + #iqUDT_Configuration.GlobalConfig.GINRangeEnd) / 2) +1;
	            END_IF;
	            "DB_GIN".GIN[#si_LastGIN110] := "DB_GIN".GIN[#iqUDT_HandshakeUpstream110.GIN];
	            //     #ts_Barcode := "DB_GIN".GIN[#iqUDT_HandshakeUpstream110.GIN].General.Identification.Barcode;
	            //     #ti_DivertDestination := "DB_GIN".GIN[#iqUDT_HandshakeUpstream110.GIN].General.SortStatus.DivertDestination;
	            #iqUDT_HandshakeUpstream110.GIN := #si_LastGIN110;

	            IF "DB_GIN".GIN[#iqUDT_HandshakeUpstream110.GIN].General.SortStatus.GoodDivert
	            THEN
	                "DB_GIN".GIN[#iqUDT_HandshakeUpstream110.GIN].WCS.ReasonCode := '1';
	            ELSE
	                "DB_GIN".GIN[#iqUDT_HandshakeUpstream110.GIN].WCS.ReasonCode := '17';
	            END_IF;


	            //     "DB_GIN".GIN[#iqUDT_HandshakeUpstream010.GIN] := "DB_GINDefault".GIN[#iqUDT_Configuration."010".PEC_EoS.DefaultGIN];
	            //     "DB_GIN".GIN[#iqUDT_HandshakeUpstream010.GIN].General.Identification.Barcode := #ts_Barcode;
	            //     "DB_GIN".GIN[#iqUDT_HandshakeUpstream010.GIN].General.SortStatus.DivertDestination := #ti_DivertDestination;

	            //     "DB_GIN".GIN[#iqUDT_HandshakeUpstream010.GIN].WCS.ReasonCode := '01';

	        END_IF;
	        IF #iqUDT_HandshakeUpstream110.GIN <> 0 THEN
	            #iqUDT_HandshakeUpstream110.GIN := #si_LastGIN110;
	        END_IF;


	    END_REGION

	    REGION Displacement
	        #sFB_Displacement110(#sUDT_Interface_110);
	    END_REGION

	    REGION Tracking

	        #sFB_Tracking_110(iUDT_ConveyorCommonConfiguration := #iqUDT_Configuration."110".Conveyor.Common,
	                          iqa_TrackingData                 := #sa_TrackingArray_110,
	                          iqUDT_ConveyorInterface          := #sUDT_Interface_110,
	                          iqUDT_HandshakeUp                := #iqUDT_HandshakeUpstream110,
	                          iqUDT_Handshake                  := #sUDT_Handshake_110);

	    END_REGION

	    REGION EoS

	        #sFB_PECUpdate_110(iUDT_PECUpdateConfiguration      := #iqUDT_Configuration."110".PEC_EoS,
	                           iUDT_ConveyorCommonConfiguration := #iqUDT_Configuration."110".Conveyor.Common,
	                           ix_PEC                           := #iUDT_MotorInput110.AllSensorPortInputs.LeftSensor,
	                           ix_TeachingMode                  := FALSE,
	                           qUDT_Status                      => #iqUDT_WorkstationStatus."110".PEC_EoS,
	                           iqUDT_ConveyorInterface          := #sUDT_Interface_110,
	                           iqUDT_UnknownGINRange            := #iqUDT_UnknownGINRange,
	                           iqUDT_FifoHeader                 := #sUDT_FifoLostGINHeaderWCS,
	                           iqUDT_Statistics                 := #iqUDT_WorkstationStatistics."110".PEC_EoS,
	                           iqa_TrackingData                 := #sa_TrackingArray_110,
	                           iqa_FifoData                     := #sa_FifoLostGINDataWCS);

	    END_REGION

	    REGION WCS lost in tracking 110
	        "FC_Fifo"(ic_Mode          := 'R',
	                  qUDT_Status      => #tudt_FifoStatus,
	                  qx_Error         => #tx_Dummy,
	                  qx_Warning       => #tx_Dummy,
	                  iqv_Data         := #ti_GIN,
	                  iqUDT_FifoHeader := #sUDT_FifoLostGINHeaderWCS,
	                  iqv_DataBuffer   := #sa_FifoLostGINDataWCS);


	        IF #ti_GIN <> 0 THEN

	            "FC_WCS_ReasonCode"(ii_GIN          := #ti_GIN,
	                                ia_Destinations := #ta_DestinationArray);

	            #sFB_DecisionUpdateWCS_110(is_PLCID            := #iqUDT_Configuration.GlobalConfig.PLCID,
	                                       is_DecisionPoint    := #iqUDT_Configuration.GlobalConfig.WCSDecisionPoint,
	                                       ii_Gin              := #ti_GIN,
	                                       iqUDT_FifoHeader    := #iqUDT_DecisionUpdateHeader,
	                                       iqa_FifoData        := #iqa_DecisionUpdateData,
	                                       iqs_Destinations    := #iqa_DecisionUpdateDestinations,
	                                       iqdi_SequenceNumber := #iqdi_DecisionUpdateSequenceNumber);



	        END_IF;

	    END_REGION

	    REGION WCS Decision update 110

	        "FC_WCS_ReasonCode"(ii_GIN          := #sa_TrackingArray_110[21],
	                            ia_Destinations := #ta_DestinationArray);

	        #sFB_DecisionUpdate_110(is_PLCID            := #iqUDT_Configuration.GlobalConfig.PLCID,
	                                is_DecisionPoint    := #iqUDT_Configuration.GlobalConfig.WCSDecisionPoint,
	                                ii_Gin              := #sa_TrackingArray_110[21],
	                                iqUDT_FifoHeader    := #iqUDT_DecisionUpdateHeader,
	                                iqa_FifoData        := #iqa_DecisionUpdateData,
	                                iqs_Destinations    := #iqa_DecisionUpdateDestinations,
	                                iqdi_SequenceNumber := #iqdi_DecisionUpdateSequenceNumber);


	    END_REGION


	    REGION Conveyor

	        #sFB_Conveyor_110(iUDT_ConveyorConfiguration := #iqUDT_Configuration."110".Conveyor,
	                          idi_PECEoSDistance         := #iqUDT_Configuration."110".PEC_EoS.Distance,
	                          idi_PECBoSDistance         := 0,
	                          ii_ExternalSpeed           := 0,
	                          ix_SafetyOk                := #ix_SafetyOk,
	                          ix_24vOk                   := #ix_24vOk,
	                          ix_400vOk                  := #ix_400vOk,
	                          ix_HardwareOk              := #iUDT_HardwareOk."110",
	                          ix_PECEoS                  := #iqUDT_WorkstationStatus."110".PEC_EoS.PEC,
	                          ix_PECBoS                  := TRUE,
	                          ix_ReverseDirection        := FALSE,
	                          ix_ExternalRequestDieBack  := (#sUDT_Interface_120.ActualSpeed = 0 AND NOT #iqUDT_WorkstationStatus."110".PEC_EoS.PEC),
	                          ix_ExternalRequestHold     := FALSE,
	                          ix_ResetEnergySave         := FALSE,
	                          qUDT_HMIStatus             => #iqUDT_WorkstationStatus."110".Conveyor,
	                          qUDT_Status                => #iqUDT_WorkstationCommonStatus."110",
	                          iqUDT_EquipmentControl     := #iqUDT_EquipmentControl,
	                          iqUDT_ConveyorCommand      := #iqUDT_WorkstationCommands."110".Conveyor,
	                          iqUDT_ConveyorInterface    := #sUDT_Interface_110,
	                          iqUDT_HandShakeUp          := #iqUDT_HandshakeUpstream110,
	                          iqUDT_HandShake            := #sUDT_Handshake_110,
	                          iqUDT_Statistics           := #iqUDT_WorkstationStatistics."110".Conveyor);

	        //  #iqUDT_HandshakeUpstream110.RTR := #iqUDT_HandshakeUpstream110.RTR AND #iqUDT_WorkstationStatus."110".PEC_EoS.PEC;


	    END_REGION

	    REGION MCO

